// TIA Portal project "Bachelor_25.04.2025_1138" (V19)

(* hardware
DEVICE "S7-1500/ET200MP station_1"  S7-1500 station
   slot 0: "Rail_0"  Rack  6ES7 590-1***0-0AA0
   slot 0: "PM 70W 120/230VAC"  PM 70W 120/230VAC  6EP1332-4BA00
   slot 1: "PLC_1"  CPU 1511-1 PN  6ES7 511-1AK00-0AB0  V1.8
      slot 3: "CPU display_1"  6ES7591-1AA00-0AA0
      slot 32768: "PROFINET interface_1"  X1
         slot 32769: "Port_1"  X1 P1
         slot 32770: "Port_2"  X1 P2
   slot 2: "DI 16x24VDC HF_1"  DI 16x24VDC HF  6ES7 521-1BH00-0AB0  V1.0
   slot 3: "DQ 16x24VDC/0.5A ST_1"  DQ 16x24VDC/0.5A ST  6ES7 522-1BH00-0AB0  V2.0
   slot 4: "AI 8xU/I/RTD/TC ST_1"  AI 8xU/I/RTD/TC ST  6ES7 531-7KF00-0AB0  V1.0
   slot 5: "AQ 4xU/I ST_1"  AQ 4xU/I ST  6ES7 532-5HD00-0AB0  V1.0
   slot 6: "CM 1542-5_1"  CM 1542-5  6GK7 542-5DX00-0XE0  V2.0
*)

// ===== PLC "PLC_1"  CPU 1511-1 PN =====

VAR_GLOBAL   // PLC tag table "Default tag table"
   "F01" AT %I0.0 : Bool;
   "F02" AT %I0.1 : Bool;
   "F11" AT %I0.2 : Bool;
   "F12" AT %I0.3 : Bool;
   "S0" AT %I0.4 : Bool;
   "PU01_AUT" AT %I0.5 : Bool;
   "PU01_MAN" AT %I0.6 : Bool;
   "PU02_AUT" AT %I1.2 : Bool;
   "PU01_RUNNING" AT %I0.7 : Bool;
   "PU01_FAULT" AT %I1.0 : Bool;
   "PU01_SS" AT %I1.1 : Bool;
   "PU02_MAN" AT %I1.3 : Bool;
   "PU02_RUNNING" AT %I1.4 : Bool;
   "PU02_FAULT" AT %I1.5 : Bool;
   "PU02_SS" AT %I1.6 : Bool;
   "FV01_GB1" AT %I1.7 : Bool;
   "FV01_GB2" AT %I2.0 : Bool;
   "FV02_GB1" AT %I2.1 : Bool;
   "FV02_GB2" AT %I2.2 : Bool;
   "PU01_RUN" AT %Q0.0 : Bool;
   "PU02_RUN" AT %Q0.1 : Bool;
   "FV01_OPEN" AT %Q0.2 : Bool;
   "FV02_OPEN" AT %Q0.3 : Bool;
   "LT01_INT" AT %IW2 : Int;
   "FT01_INT" AT %IW10 : Int;
   "FT02_INT" AT %IW4 : Int;
   "PU01_INT" AT %QW2 : Int;
   "PU02_INT" AT %QW4 : Int;
   "M_F01" AT %M0.0 : Bool;
   "M_F02" AT %M0.1 : Bool;
   "M_F11" AT %M0.2 : Bool;
   "M_F12" AT %M0.3 : Bool;
   "M_S0" AT %M0.4 : Bool;
   "M_PU01_AUT" AT %M0.5 : Bool;
   "M_PU01_MAN" AT %M0.6 : Bool;
   "M_PU01_RUNNING" AT %M0.7 : Bool;
   "M_PU01_FAULT" AT %M2.0 : Bool;
   "M_PU01_SS" AT %M2.1 : Bool;
   "M_PU02_AUT" AT %M2.2 : Bool;
   "M_PU02_MAN" AT %M2.3 : Bool;
   "M_PU02_RUNNING" AT %M2.4 : Bool;
   "M_PU02_FAULT" AT %M2.5 : Bool;
   "M_PU02_SS" AT %M2.6 : Bool;
   "M_FV01_GB1" AT %M2.7 : Bool;
   "M_FV01_GB2" AT %M3.0 : Bool;
   "M_FV02_GB1" AT %M3.1 : Bool;
   "M_FV02_GB2" AT %M3.2 : Bool;
   "M_PU01_RUN" AT %M4.0 : Bool;
   "M_PU02_RUN" AT %M4.1 : Bool;
   "M_FV01" AT %M4.2 : Bool;
   "M_FV02" AT %M4.3 : Bool;
   "PU01_REAL" AT %MD100 : Real;
   "PU02_REAL" AT %MD104 : Real;
   "LT01_REAL" AT %MD108 : Real;
   "FT01_REAL" AT %MD1120 : Real;
   "FT02_REAL" AT %MD116 : Real;
   "RESET" AT %I2.3 : Bool;
   "Tag_1" AT %MW200 : Int;
   "Tag_21" AT %MW204 : Int;
   "Tag_22" AT %MW208 : Int;
   "Tag_23" AT %MW212 : Int;
   "Tag_24" AT %MW216 : Int;
   "BEST_HOURS" AT %MD50 : DInt;
   "OPTIMAL_HOUR" AT %M5.0 : Bool;
   "Tag_2" AT %MW300 : Word;
   "Tag_3" AT %MD320 : Real;
   "TRANSMIT" AT %I6.0 : "transmitter_dt";
   "CONTROLLER_STATE" AT %MW220 : Int;
   "M_PU01_AUT_SCADA" AT %M1000.0 : Bool;
   "M_PU01_MAN_SCADA" AT %M1.1 : Bool;
   "M_PU02_AUT_SCADA" AT %M1000.1 : Bool;
   "M_PU02_MAN_SCADA" AT %M3.4 : Bool;
   "ALWAYS HIGH" AT %M1.2 : Bool;
   "ALWAYS LOW" AT %M1.3 : Bool;
   "Clock_Byte" AT %MB6 : Byte;
   "Clock_10Hz" AT %M6.0 : Bool;
   "Clock_5Hz" AT %M6.1 : Bool;
   "Clock_2.5Hz" AT %M6.2 : Bool;
   "Clock_2Hz" AT %M6.3 : Bool;
   "Clock_1.25Hz" AT %M6.4 : Bool;
   "Clock_1Hz" AT %M6.5 : Bool;
   "Clock_0.625Hz" AT %M6.6 : Bool;
   "Clock_0.5Hz" AT %M6.7 : Bool;
   "BEST_HOURS_DAG2" AT %MD60 : DInt;
END_VAR

TYPE "transmitter_dt"
   STRUCT
      test_1 : Bool;
      test_2 : Bool;
      test_3 : Int;
   END_STRUCT;
END_TYPE

// folder: Data Blocks

DATA_BLOCK "FT02_DB"   // DB1
{ S7_Optimized_Access := 'FALSE' }
VERSION : 0.1
// stored: InstanceOfName Transmitter
"Transmitter"
BEGIN
   t_sp_hh_pct := 100.0;
   t_sp_h_pct := 100.0;
   t_sp_l_pct := 0.0;
   t_sp_ll_pct := 0.0;
   t_sp_scale_high_pct := 100.0;
END_DATA_BLOCK

DATA_BLOCK "Cascade Regulator_DB"   // DB2
{ S7_Optimized_Access := 'FALSE' }
VERSION : 0.1
// stored: InstanceOfName Cascade Regulator
"Cascade Regulator"
BEGIN
END_DATA_BLOCK

DATA_BLOCK "PU02_DB"   // DB3
{ S7_Optimized_Access := 'FALSE' }
VERSION : 0.1
// stored: InstanceOfName Pump
"Pump"
BEGIN
END_DATA_BLOCK

DATA_BLOCK "LT01_DB"   // DB5
{ S7_Optimized_Access := 'FALSE' }
VERSION : 0.1
// stored: InstanceOfName Transmitter
"Transmitter"
BEGIN
   t_hys := 1;
   t_sp_hh_pct := 95.0;
   t_sp_h_pct := 90.0;
   t_sp_l_pct := 30.0;
   t_sp_ll_pct := 25.0;
   t_sp_scale_high_pct := 100.0;
   t_sp_scale_high_sca := 4.0;
   t_sp_hh_sca := 3.8;
   t_sp_h_sca := 3.6;
   t_sp_l_sca := 0.9;
   t_sp_ll_sca := 0.6;
END_DATA_BLOCK

DATA_BLOCK "FT01_DB"   // DB6
{ S7_Optimized_Access := 'FALSE' }
VERSION : 0.1
// stored: InstanceOfName Transmitter
"Transmitter"
BEGIN
   t_sp_hh_pct := 100.0;
   t_sp_h_pct := 100.0;
   t_sp_l_pct := 0.0;
   t_sp_ll_pct := 0.0;
   t_sp_scale_high_pct := 100.0;
   t_sp_scale_high_sca := 50.0;
   t_sp_hh_sca := 50.0;
   t_sp_h_sca := 50.0;
END_DATA_BLOCK

DATA_BLOCK "Control_block_DB"   // DB7
{ S7_Optimized_Access := 'FALSE' }
VERSION : 0.1
// stored: InstanceOfName Control block
"Control block"
BEGIN
END_DATA_BLOCK

DATA_BLOCK "PU01_DB"   // DB14
{ S7_Optimized_Access := 'FALSE' }
VERSION : 0.1
// stored: InstanceOfName Pump
"Pump"
BEGIN
END_DATA_BLOCK

DATA_BLOCK "Check optimal hour 48h_DB"   // DB29
{ S7_Optimized_Access := 'TRUE' }
VERSION : 0.1
// stored: InstanceOfName Check optimal hour 48h
"Check optimal hour 48h"
BEGIN
END_DATA_BLOCK

// folder: System blocks/Program resources

DATA_BLOCK "IEC_Timer_0_DB"   // DB4
{ S7_Optimized_Access := 'TRUE' }
AUTHOR : Simatic
FAMILY : IEC
NAME : IEC_TMR
VERSION : 1.0
// stored: InstanceOfName IEC_TIMER
"IEC_TIMER"
BEGIN
END_DATA_BLOCK

DATA_BLOCK "t_alarm_hys"   // DB8
{ S7_Optimized_Access := 'TRUE' }
AUTHOR : Simatic
FAMILY : IEC
NAME : IEC_TMR
VERSION : 1.0
// stored: InstanceOfName IEC_TIMER
"IEC_TIMER"
BEGIN
END_DATA_BLOCK

DATA_BLOCK "IEC_Timer_0_DB_2"   // DB11
{ S7_Optimized_Access := 'TRUE' }
AUTHOR : Simatic
FAMILY : IEC
NAME : IEC_TMR
VERSION : 1.0
// stored: InstanceOfName IEC_TIMER
"IEC_TIMER"
BEGIN
END_DATA_BLOCK

DATA_BLOCK "t_alarm_hh"   // DB12
{ S7_Optimized_Access := 'TRUE' }
AUTHOR : Simatic
FAMILY : IEC
NAME : IEC_TMR
VERSION : 1.0
// stored: InstanceOfName IEC_TIMER
"IEC_TIMER"
BEGIN
END_DATA_BLOCK

DATA_BLOCK "t_alarm_h"   // DB13
{ S7_Optimized_Access := 'TRUE' }
AUTHOR : Simatic
FAMILY : IEC
NAME : IEC_TMR
VERSION : 1.0
// stored: InstanceOfName IEC_TIMER
"IEC_TIMER"
BEGIN
END_DATA_BLOCK

DATA_BLOCK "t_alarm_l"   // DB15
{ S7_Optimized_Access := 'TRUE' }
AUTHOR : Simatic
FAMILY : IEC
NAME : IEC_TMR
VERSION : 1.0
// stored: InstanceOfName IEC_TIMER
"IEC_TIMER"
BEGIN
END_DATA_BLOCK

DATA_BLOCK "t_alarm_ll"   // DB16
{ S7_Optimized_Access := 'TRUE' }
AUTHOR : Simatic
FAMILY : IEC
NAME : IEC_TMR
VERSION : 1.0
// stored: InstanceOfName IEC_TIMER
"IEC_TIMER"
BEGIN
END_DATA_BLOCK

DATA_BLOCK "t_alarm_range"   // DB17
{ S7_Optimized_Access := 'TRUE' }
AUTHOR : Simatic
FAMILY : IEC
NAME : IEC_TMR
VERSION : 1.0
// stored: InstanceOfName IEC_TIMER
"IEC_TIMER"
BEGIN
END_DATA_BLOCK

DATA_BLOCK "p_alarm_fv"   // DB18
{ S7_Optimized_Access := 'TRUE' }
AUTHOR : Simatic
FAMILY : IEC
NAME : IEC_TMR
VERSION : 1.0
// stored: InstanceOfName IEC_TIMER
"IEC_TIMER"
BEGIN
END_DATA_BLOCK

DATA_BLOCK "p_alarm_vfd"   // DB19
{ S7_Optimized_Access := 'TRUE' }
AUTHOR : Simatic
FAMILY : IEC
NAME : IEC_TMR
VERSION : 1.0
// stored: InstanceOfName IEC_TIMER
"IEC_TIMER"
BEGIN
END_DATA_BLOCK

DATA_BLOCK "p_alarm_tmp"   // DB20
{ S7_Optimized_Access := 'TRUE' }
AUTHOR : Simatic
FAMILY : IEC
NAME : IEC_TMR
VERSION : 1.0
// stored: InstanceOfName IEC_TIMER
"IEC_TIMER"
BEGIN
END_DATA_BLOCK

DATA_BLOCK "p_alarm_moi"   // DB21
{ S7_Optimized_Access := 'TRUE' }
AUTHOR : Simatic
FAMILY : IEC
NAME : IEC_TMR
VERSION : 1.0
// stored: InstanceOfName IEC_TIMER
"IEC_TIMER"
BEGIN
END_DATA_BLOCK

DATA_BLOCK "p_alarm"   // DB22
{ S7_Optimized_Access := 'TRUE' }
AUTHOR : Simatic
FAMILY : IEC
NAME : IEC_TMR
VERSION : 1.0
// stored: InstanceOfName IEC_TIMER
"IEC_TIMER"
BEGIN
END_DATA_BLOCK

DATA_BLOCK "Input Error"   // DB23
{ S7_Optimized_Access := 'TRUE' }
AUTHOR : Simatic
FAMILY : IEC
NAME : IEC_TMR
VERSION : 1.0
// stored: InstanceOfName IEC_TIMER
"IEC_TIMER"
BEGIN
END_DATA_BLOCK

DATA_BLOCK "Tuning Error"   // DB24
{ S7_Optimized_Access := 'TRUE' }
AUTHOR : Simatic
FAMILY : IEC
NAME : IEC_TMR
VERSION : 1.0
// stored: InstanceOfName IEC_TIMER
"IEC_TIMER"
BEGIN
END_DATA_BLOCK

DATA_BLOCK "Setpoint Error"   // DB25
{ S7_Optimized_Access := 'TRUE' }
AUTHOR : Simatic
FAMILY : IEC
NAME : IEC_TMR
VERSION : 1.0
// stored: InstanceOfName IEC_TIMER
"IEC_TIMER"
BEGIN
END_DATA_BLOCK

DATA_BLOCK "ManualValue Error"   // DB26
{ S7_Optimized_Access := 'TRUE' }
AUTHOR : Simatic
FAMILY : IEC
NAME : IEC_TMR
VERSION : 1.0
// stored: InstanceOfName IEC_TIMER
"IEC_TIMER"
BEGIN
END_DATA_BLOCK

DATA_BLOCK "General Error"   // DB27
{ S7_Optimized_Access := 'TRUE' }
AUTHOR : Simatic
FAMILY : IEC
NAME : IEC_TMR
VERSION : 1.0
// stored: InstanceOfName IEC_TIMER
"IEC_TIMER"
BEGIN
END_DATA_BLOCK

DATA_BLOCK "Regulator Error"   // DB28
{ S7_Optimized_Access := 'TRUE' }
AUTHOR : Simatic
FAMILY : IEC
NAME : IEC_TMR
VERSION : 1.0
// stored: InstanceOfName IEC_TIMER
"IEC_TIMER"
BEGIN
END_DATA_BLOCK

DATA_BLOCK "CV_unmod"   // DB30
{ S7_Optimized_Access := 'TRUE' }
AUTHOR : Simatic
FAMILY : IEC
NAME : IEC_TMR
VERSION : 1.0
// stored: InstanceOfName IEC_TIMER
"IEC_TIMER"
BEGIN
END_DATA_BLOCK

DATA_BLOCK "Timer"   // DB31
{ S7_Optimized_Access := 'TRUE' }
AUTHOR : Simatic
FAMILY : IEC
NAME : IEC_TMR
VERSION : 1.0
// stored: InstanceOfName IEC_TIMER
"IEC_TIMER"
BEGIN
END_DATA_BLOCK

DATA_BLOCK "p_alarm_flow"   // DB32
{ S7_Optimized_Access := 'TRUE' }
AUTHOR : Simatic
FAMILY : IEC
NAME : IEC_TMR
VERSION : 1.0
// stored: InstanceOfName IEC_TIMER
"IEC_TIMER"
BEGIN
END_DATA_BLOCK

// folder: (top level)

FUNCTION_BLOCK "Control block"   // FB1, LAD
{ S7_Optimized_Access := 'FALSE' }
VERSION : 0.1
   VAR_INPUT
      pu01_aut : Bool;
      pu01_aut_scada : Bool := true;
      pu01_man : Bool;
      pu01_man_scada : Bool;
      pu01_mv : Real;
      pu01_fault : Bool;
      pu02_aut : Bool;
      pu02_aut_scada : Bool := true;
      pu02_man : Bool;
      pu02_man_scada : Bool;
      pu02_mv : Real;
      pu02_fault : Bool;
      setpoint_high : Real;
      setpoint_low : Real;
      controller_cv : Real;
      pump_time : Time := T#30s;
   END_VAR
   VAR_OUTPUT
      controller_state : Int;
      controller_mv : Real;
   END_VAR
   VAR_IN_OUT
      pu01_run : Bool;
      pu01_running : Bool;
      pu02_run : Bool;
      pu02_running : Bool;
   END_VAR
   VAR
      "pu01 is in aut" : Bool;
      "pu01 is in man" : Bool;
      "pu02 is in aut" : Bool;
      "pu02 is in man" : Bool;
      yup : Int;
      yupper : Bool;
      n_trig_0 : Bool;
      n_trig_1 : Bool;
      n_trig_2 : Bool;
      n_trig_3 : Bool;
      pu01_timer : Time := T#30s;
      pu02_timer : Time := T#40s;
   END_VAR
   VAR_TEMP   // added for the SCL form of the ladder/FBD networks
      _w1 : Bool;
      _w2 : Bool;
   END_VAR
BEGIN

REGION Network 1: PU01 Automatic
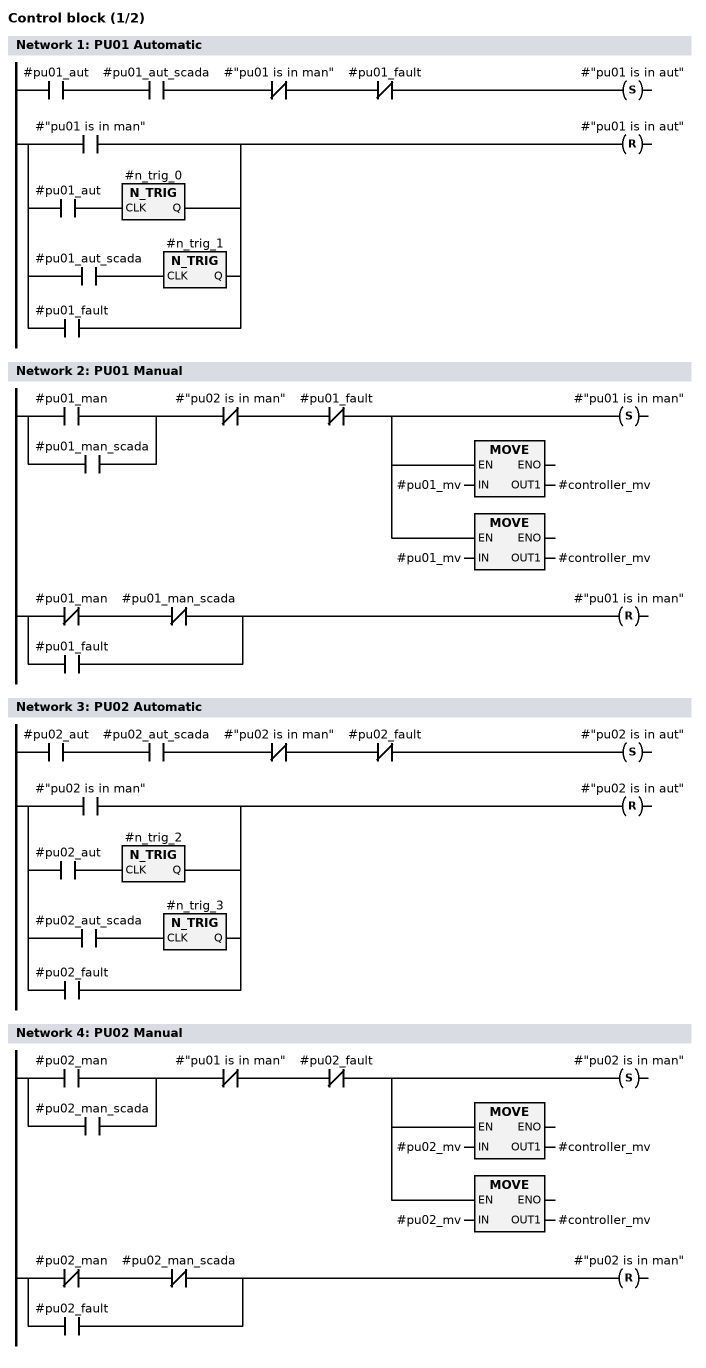
   RUNG wire#powerrail
      Contact( #pu01_aut )
      Contact( #pu01_aut_scada )
      I_Contact( #"pu01 is in man" )
      I_Contact( #pu01_fault )
      S_Coil( #"pu01 is in aut" )
   END_RUNG
   RUNG wire#powerrail
      Contact( #"pu01 is in man" )
      wire#w1
      R_Coil( #"pu01 is in aut" )
   END_RUNG
   RUNG wire#powerrail
      Contact( #pu01_aut )
      N_Trig( #n_trig_0 )
   END_RUNG wire#w1
   RUNG wire#powerrail
      Contact( #pu01_aut_scada )
      N_Trig( #n_trig_1 )
   END_RUNG wire#w1
   RUNG wire#powerrail
      Contact( #pu01_fault )
   END_RUNG wire#w1
   // the same network as SCL:
   IF #pu01_aut AND #pu01_aut_scada AND NOT #"pu01 is in man" AND NOT #pu01_fault THEN
       #"pu01 is in aut" := TRUE;
   END_IF;
   #_w1 := NOT #pu01_aut AND #n_trig_0;   // falling edge
   #n_trig_0 := #pu01_aut;
   #_w2 := NOT #pu01_aut_scada AND #n_trig_1;   // falling edge
   #n_trig_1 := #pu01_aut_scada;
   IF #"pu01 is in man" OR #_w1 OR #_w2 OR #pu01_fault THEN #"pu01 is in aut" := FALSE; END_IF;
END_REGION

REGION Network 2: PU01 Manual
   RUNG wire#powerrail
      Contact( #pu01_man )
      wire#w1
      I_Contact( #"pu02 is in man" )
      I_Contact( #pu01_fault )
      wire#w2
      S_Coil( #"pu01 is in man" )
   END_RUNG
   RUNG wire#powerrail
      Contact( #pu01_man_scada )
   END_RUNG wire#w1
   RUNG wire#w2
      Move(in := #pu01_mv, out1 => #controller_mv)
   END_RUNG
   RUNG wire#w2
      Move(in := #pu01_mv, out1 => #controller_mv)
   END_RUNG
   RUNG wire#powerrail
      I_Contact( #pu01_man )
      I_Contact( #pu01_man_scada )
      wire#w3
      R_Coil( #"pu01 is in man" )
   END_RUNG
   RUNG wire#powerrail
      Contact( #pu01_fault )
   END_RUNG wire#w3
   // the same network as SCL:
   IF (#pu01_man OR #pu01_man_scada) AND NOT #"pu02 is in man" AND NOT #pu01_fault THEN
       #"pu01 is in man" := TRUE;
       #controller_mv := #pu01_mv;
       #controller_mv := #pu01_mv;
   END_IF;
   IF (NOT #pu01_man AND NOT #pu01_man_scada) OR #pu01_fault THEN #"pu01 is in man" := FALSE; END_IF;
END_REGION

REGION Network 3: PU02 Automatic
   RUNG wire#powerrail
      Contact( #pu02_aut )
      Contact( #pu02_aut_scada )
      I_Contact( #"pu02 is in man" )
      I_Contact( #pu02_fault )
      S_Coil( #"pu02 is in aut" )
   END_RUNG
   RUNG wire#powerrail
      Contact( #"pu02 is in man" )
      wire#w1
      R_Coil( #"pu02 is in aut" )
   END_RUNG
   RUNG wire#powerrail
      Contact( #pu02_aut )
      N_Trig( #n_trig_2 )
   END_RUNG wire#w1
   RUNG wire#powerrail
      Contact( #pu02_aut_scada )
      N_Trig( #n_trig_3 )
   END_RUNG wire#w1
   RUNG wire#powerrail
      Contact( #pu02_fault )
   END_RUNG wire#w1
   // the same network as SCL:
   IF #pu02_aut AND #pu02_aut_scada AND NOT #"pu02 is in man" AND NOT #pu02_fault THEN
       #"pu02 is in aut" := TRUE;
   END_IF;
   #_w1 := NOT #pu02_aut AND #n_trig_2;   // falling edge
   #n_trig_2 := #pu02_aut;
   #_w2 := NOT #pu02_aut_scada AND #n_trig_3;   // falling edge
   #n_trig_3 := #pu02_aut_scada;
   IF #"pu02 is in man" OR #_w1 OR #_w2 OR #pu02_fault THEN #"pu02 is in aut" := FALSE; END_IF;
END_REGION

REGION Network 4: PU02 Manual
   RUNG wire#powerrail
      Contact( #pu02_man )
      wire#w1
      I_Contact( #"pu01 is in man" )
      I_Contact( #pu02_fault )
      wire#w2
      S_Coil( #"pu02 is in man" )
   END_RUNG
   RUNG wire#powerrail
      Contact( #pu02_man_scada )
   END_RUNG wire#w1
   RUNG wire#w2
      Move(in := #pu02_mv, out1 => #controller_mv)
   END_RUNG
   RUNG wire#w2
      Move(in := #pu02_mv, out1 => #controller_mv)
   END_RUNG
   RUNG wire#powerrail
      I_Contact( #pu02_man )
      I_Contact( #pu02_man_scada )
      wire#w3
      R_Coil( #"pu02 is in man" )
   END_RUNG
   RUNG wire#powerrail
      Contact( #pu02_fault )
   END_RUNG wire#w3
   // the same network as SCL:
   IF (#pu02_man OR #pu02_man_scada) AND NOT #"pu01 is in man" AND NOT #pu02_fault THEN
       #"pu02 is in man" := TRUE;
       #controller_mv := #pu02_mv;
       #controller_mv := #pu02_mv;
   END_IF;
   IF (NOT #pu02_man AND NOT #pu02_man_scada) OR #pu02_fault THEN #"pu02 is in man" := FALSE; END_IF;
END_REGION

REGION Network 5: Controller Auto
   // Sets the Controller in auto if it can.
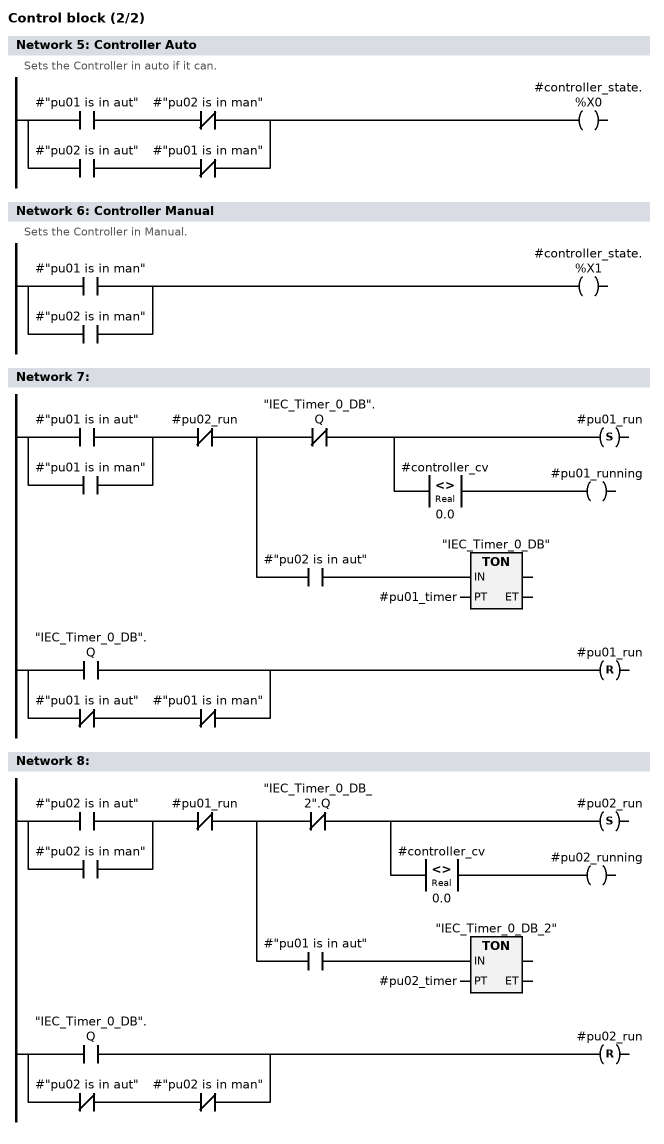
   RUNG wire#powerrail
      Contact( #"pu01 is in aut" )
      I_Contact( #"pu02 is in man" )
      wire#w1
      Coil( #controller_state.%X0 )
   END_RUNG
   RUNG wire#powerrail
      Contact( #"pu02 is in aut" )
      I_Contact( #"pu01 is in man" )
   END_RUNG wire#w1
   // the same network as SCL:
   #controller_state.%X0 := (#"pu01 is in aut" AND NOT #"pu02 is in man") OR (#"pu02 is in aut" AND NOT #"pu01 is in man");
END_REGION

REGION Network 6: Controller Manual
   // Sets the Controller in Manual.
   RUNG wire#powerrail
      Contact( #"pu01 is in man" )
      wire#w1
      Coil( #controller_state.%X1 )
   END_RUNG
   RUNG wire#powerrail
      Contact( #"pu02 is in man" )
   END_RUNG wire#w1
   // the same network as SCL:
   #controller_state.%X1 := #"pu01 is in man" OR #"pu02 is in man";
END_REGION

REGION Network 7
   #_w1 := (#"pu01 is in aut" OR #"pu01 is in man") AND NOT #pu02_run;
   #_w2 := #_w1 AND NOT "IEC_Timer_0_DB".Q;
   IF #_w2 THEN #pu01_run := TRUE; END_IF;
   #pu01_running := #_w2 AND (#controller_cv <> 0.0);
   "IEC_Timer_0_DB".TON(IN := #_w1 AND #"pu02 is in aut", PT := #pu01_timer);
   IF "IEC_Timer_0_DB".Q OR (NOT #"pu01 is in aut" AND NOT #"pu01 is in man") THEN
       #pu01_run := FALSE;
   END_IF;
END_REGION

REGION Network 8
   #_w1 := (#"pu02 is in aut" OR #"pu02 is in man") AND NOT #pu01_run;
   #_w2 := #_w1 AND NOT "IEC_Timer_0_DB_2".Q;
   IF #_w2 THEN #pu02_run := TRUE; END_IF;
   #pu02_running := #_w2 AND (#controller_cv <> 0.0);
   "IEC_Timer_0_DB_2".TON(IN := #_w1 AND #"pu01 is in aut", PT := #pu02_timer);
   IF "IEC_Timer_0_DB".Q OR (NOT #"pu02 is in aut" AND NOT #"pu02 is in man") THEN
       #pu02_run := FALSE;
   END_IF;
END_REGION
END_FUNCTION_BLOCK

FUNCTION "Convert Analog Values" : Void   // FC1, LAD
{ S7_Optimized_Access := 'TRUE' }
VERSION : 0.1
   VAR_INPUT
      lt01_int : Int;
      ft01_int : Int;
      ft02_int : Int;
      pu01_real : Real;
      pu02_real : Real;
   END_VAR
   VAR_OUTPUT
      lt01_real : Real;
      ft01_real : Real;
      ft02_real : Real;
      pu01_int : Int;
      pu02_int : Int;
   END_VAR
   VAR_TEMP
      lt01_temp : Real;
      ft01_temp : Real;
      ft02_temp : Real;
      pu01_temp : Real;
      pu02_temp : Real;
   END_VAR
BEGIN

REGION Network 1: Level Transmitter 01
   // Level Transmitter in the pool
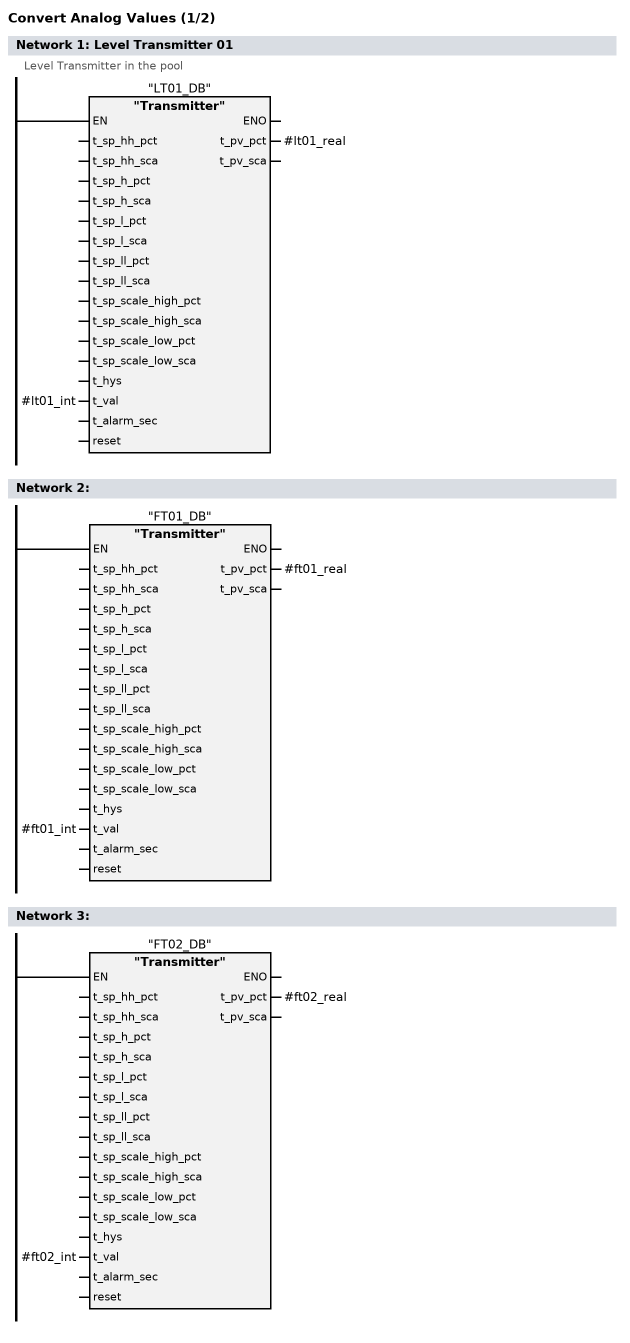
   RUNG wire#powerrail
      "LT01_DB"(t_sp_hh_pct :=, t_sp_hh_sca :=, t_sp_h_pct :=, t_sp_h_sca :=, t_sp_l_pct :=, t_sp_l_sca :=, t_sp_ll_pct :=, t_sp_ll_sca :=, t_sp_scale_high_pct :=, t_sp_scale_high_sca :=, t_sp_scale_low_pct :=, t_sp_scale_low_sca :=, t_hys :=, t_val := #lt01_int, t_alarm_sec :=, reset :=, t_pv_pct => #lt01_real, t_pv_sca =>)
   END_RUNG
   // the same network as SCL:
   "LT01_DB"(t_val := #lt01_int, t_pv_pct => #lt01_real);   // "Transmitter"
END_REGION

REGION Network 2
   RUNG wire#powerrail
      "FT01_DB"(t_sp_hh_pct :=, t_sp_hh_sca :=, t_sp_h_pct :=, t_sp_h_sca :=, t_sp_l_pct :=, t_sp_l_sca :=, t_sp_ll_pct :=, t_sp_ll_sca :=, t_sp_scale_high_pct :=, t_sp_scale_high_sca :=, t_sp_scale_low_pct :=, t_sp_scale_low_sca :=, t_hys :=, t_val := #ft01_int, t_alarm_sec :=, reset :=, t_pv_pct => #ft01_real, t_pv_sca =>)
   END_RUNG
   // the same network as SCL:
   "FT01_DB"(t_val := #ft01_int, t_pv_pct => #ft01_real);   // "Transmitter"
END_REGION

REGION Network 3
   RUNG wire#powerrail
      "FT02_DB"(t_sp_hh_pct :=, t_sp_hh_sca :=, t_sp_h_pct :=, t_sp_h_sca :=, t_sp_l_pct :=, t_sp_l_sca :=, t_sp_ll_pct :=, t_sp_ll_sca :=, t_sp_scale_high_pct :=, t_sp_scale_high_sca :=, t_sp_scale_low_pct :=, t_sp_scale_low_sca :=, t_hys :=, t_val := #ft02_int, t_alarm_sec :=, reset :=, t_pv_pct => #ft02_real, t_pv_sca =>)
   END_RUNG
   // the same network as SCL:
   "FT02_DB"(t_val := #ft02_int, t_pv_pct => #ft02_real);   // "Transmitter"
END_REGION

REGION Network 4: Signal til frekvensomformeren som tilhører PU01
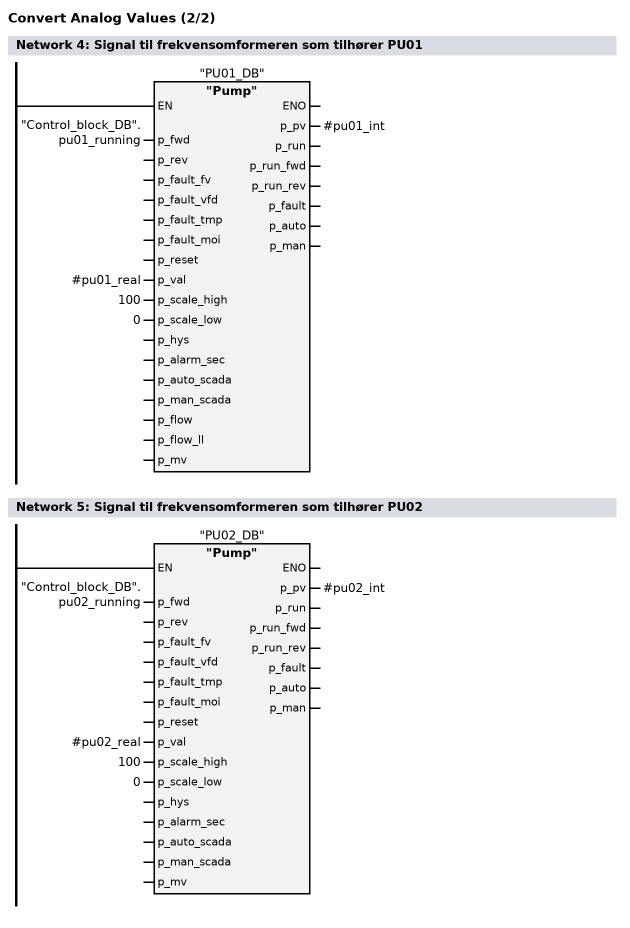
   RUNG wire#powerrail
      "PU01_DB"(p_fwd := "Control_block_DB".pu01_running, p_rev :=, p_fault_fv :=, p_fault_vfd :=, p_fault_tmp :=, p_fault_moi :=, p_reset :=, p_val := #pu01_real, p_scale_high := 100, p_scale_low := 0, p_hys :=, p_alarm_sec :=, p_auto_scada :=, p_man_scada :=, p_flow :=, p_flow_ll :=, p_mv :=, p_pv => #pu01_int, p_run =>, p_run_fwd =>, p_run_rev =>, p_fault =>, p_auto =>, p_man =>)
   END_RUNG
   // the same network as SCL:
   "PU01_DB"(p_fwd := "Control_block_DB".pu01_running,   // "Pump"
             p_val := #pu01_real,
             p_scale_high := 100,
             p_scale_low := 0,
             p_pv => #pu01_int);
END_REGION

REGION Network 5: Signal til frekvensomformeren som tilhører PU02
   RUNG wire#powerrail
      "PU02_DB"(p_fwd := "Control_block_DB".pu02_running, p_rev :=, p_fault_fv :=, p_fault_vfd :=, p_fault_tmp :=, p_fault_moi :=, p_reset :=, p_val := #pu02_real, p_scale_high := 100, p_scale_low := 0, p_hys :=, p_alarm_sec :=, p_auto_scada :=, p_man_scada :=, p_mv :=, p_pv => #pu02_int, p_run =>, p_run_fwd =>, p_run_rev =>, p_fault =>, p_auto =>, p_man =>)
   END_RUNG
   // the same network as SCL:
   "PU02_DB"(p_fwd := "Control_block_DB".pu02_running,   // "Pump"
             p_val := #pu02_real,
             p_scale_high := 100,
             p_scale_low := 0,
             p_pv => #pu02_int);
END_REGION
END_FUNCTION

FUNCTION "Input Mapping" : Void   // FC3, LAD
TITLE = Convert I/O to M
{ S7_Optimized_Access := 'TRUE' }
VERSION : 0.1
BEGIN

REGION Network 1: Digital Inputs
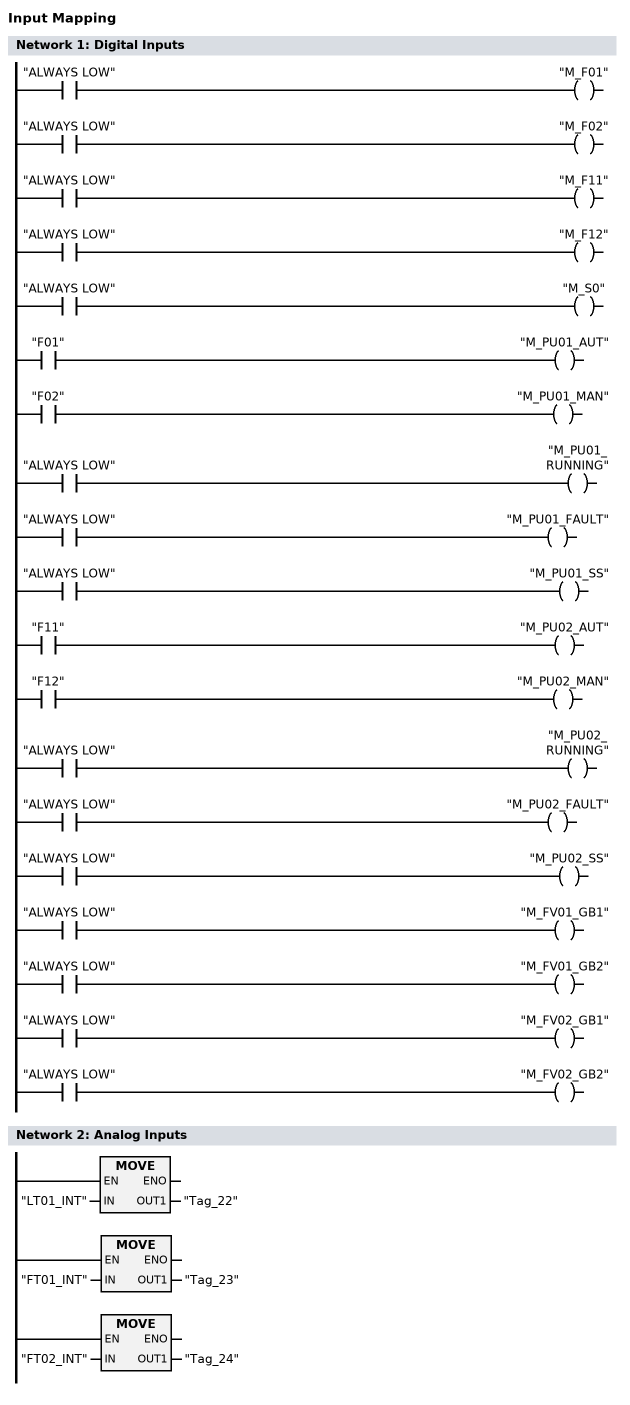
   RUNG wire#powerrail
      Contact( "ALWAYS LOW" )
      Coil( "M_F01" )
   END_RUNG
   RUNG wire#powerrail
      Contact( "ALWAYS LOW" )
      Coil( "M_F02" )
   END_RUNG
   RUNG wire#powerrail
      Contact( "ALWAYS LOW" )
      Coil( "M_F11" )
   END_RUNG
   RUNG wire#powerrail
      Contact( "ALWAYS LOW" )
      Coil( "M_F12" )
   END_RUNG
   RUNG wire#powerrail
      Contact( "ALWAYS LOW" )
      Coil( "M_S0" )
   END_RUNG
   RUNG wire#powerrail
      Contact( "F01" )
      Coil( "M_PU01_AUT" )
   END_RUNG
   RUNG wire#powerrail
      Contact( "F02" )
      Coil( "M_PU01_MAN" )
   END_RUNG
   RUNG wire#powerrail
      Contact( "ALWAYS LOW" )
      Coil( "M_PU01_RUNNING" )
   END_RUNG
   RUNG wire#powerrail
      Contact( "ALWAYS LOW" )
      Coil( "M_PU01_FAULT" )
   END_RUNG
   RUNG wire#powerrail
      Contact( "ALWAYS LOW" )
      Coil( "M_PU01_SS" )
   END_RUNG
   RUNG wire#powerrail
      Contact( "F11" )
      Coil( "M_PU02_AUT" )
   END_RUNG
   RUNG wire#powerrail
      Contact( "F12" )
      Coil( "M_PU02_MAN" )
   END_RUNG
   RUNG wire#powerrail
      Contact( "ALWAYS LOW" )
      Coil( "M_PU02_RUNNING" )
   END_RUNG
   RUNG wire#powerrail
      Contact( "ALWAYS LOW" )
      Coil( "M_PU02_FAULT" )
   END_RUNG
   RUNG wire#powerrail
      Contact( "ALWAYS LOW" )
      Coil( "M_PU02_SS" )
   END_RUNG
   RUNG wire#powerrail
      Contact( "ALWAYS LOW" )
      Coil( "M_FV01_GB1" )
   END_RUNG
   RUNG wire#powerrail
      Contact( "ALWAYS LOW" )
      Coil( "M_FV01_GB2" )
   END_RUNG
   RUNG wire#powerrail
      Contact( "ALWAYS LOW" )
      Coil( "M_FV02_GB1" )
   END_RUNG
   RUNG wire#powerrail
      Contact( "ALWAYS LOW" )
      Coil( "M_FV02_GB2" )
   END_RUNG
   // the same network as SCL:
   "M_F01" := "ALWAYS LOW";
   "M_F02" := "ALWAYS LOW";
   "M_F11" := "ALWAYS LOW";
   "M_F12" := "ALWAYS LOW";
   "M_S0" := "ALWAYS LOW";
   "M_PU01_AUT" := "F01";
   "M_PU01_MAN" := "F02";
   "M_PU01_RUNNING" := "ALWAYS LOW";
   "M_PU01_FAULT" := "ALWAYS LOW";
   "M_PU01_SS" := "ALWAYS LOW";
   "M_PU02_AUT" := "F11";
   "M_PU02_MAN" := "F12";
   "M_PU02_RUNNING" := "ALWAYS LOW";
   "M_PU02_FAULT" := "ALWAYS LOW";
   "M_PU02_SS" := "ALWAYS LOW";
   "M_FV01_GB1" := "ALWAYS LOW";
   "M_FV01_GB2" := "ALWAYS LOW";
   "M_FV02_GB1" := "ALWAYS LOW";
   "M_FV02_GB2" := "ALWAYS LOW";
END_REGION

REGION Network 2: Analog Inputs
   RUNG wire#powerrail
      Move(in := "LT01_INT", out1 => "Tag_22")
   END_RUNG
   RUNG wire#powerrail
      Move(in := "FT01_INT", out1 => "Tag_23")
   END_RUNG
   RUNG wire#powerrail
      Move(in := "FT02_INT", out1 => "Tag_24")
   END_RUNG
   // the same network as SCL:
   "Tag_22" := "LT01_INT";
   "Tag_23" := "FT01_INT";
   "Tag_24" := "FT02_INT";
END_REGION
END_FUNCTION

FUNCTION "Output Mapping" : Void   // FC4, LAD
{ S7_Optimized_Access := 'TRUE' }
VERSION : 0.1
BEGIN

REGION Network 1: Digital Outputs
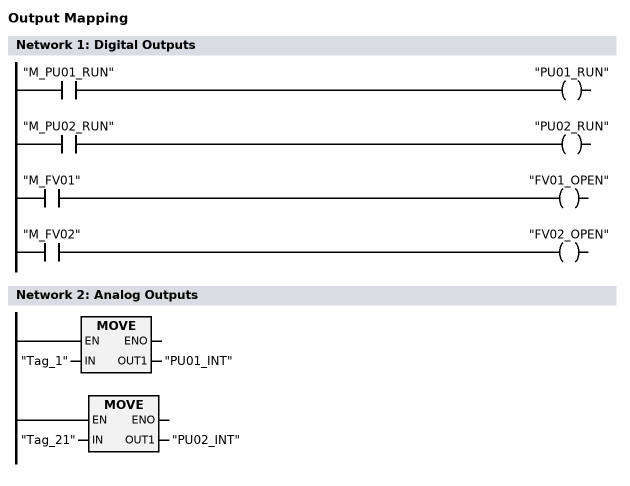
   RUNG wire#powerrail
      Contact( "M_PU01_RUN" )
      Coil( "PU01_RUN" )
   END_RUNG
   RUNG wire#powerrail
      Contact( "M_PU02_RUN" )
      Coil( "PU02_RUN" )
   END_RUNG
   RUNG wire#powerrail
      Contact( "M_FV01" )
      Coil( "FV01_OPEN" )
   END_RUNG
   RUNG wire#powerrail
      Contact( "M_FV02" )
      Coil( "FV02_OPEN" )
   END_RUNG
   // the same network as SCL:
   "PU01_RUN" := "M_PU01_RUN";
   "PU02_RUN" := "M_PU02_RUN";
   "FV01_OPEN" := "M_FV01";
   "FV02_OPEN" := "M_FV02";
END_REGION

REGION Network 2: Analog Outputs
   RUNG wire#powerrail
      Move(in := "Tag_1", out1 => "PU01_INT")
   END_RUNG
   RUNG wire#powerrail
      Move(in := "Tag_21", out1 => "PU02_INT")
   END_RUNG
   // the same network as SCL:
   "PU01_INT" := "Tag_1";
   "PU02_INT" := "Tag_21";
END_REGION
END_FUNCTION

ORGANIZATION_BLOCK "Main"   // OB1, LAD, ProgramCycle
TITLE = "Main Program Sweep (Cycle)"
{ S7_Optimized_Access := 'TRUE' }
VERSION : 0.1
   VAR_INPUT
      Initial_Call : Bool;   // Initial call of this OB
      Remanence : Bool;   // =True, if remanent data are available
   END_VAR
BEGIN

REGION Network 1
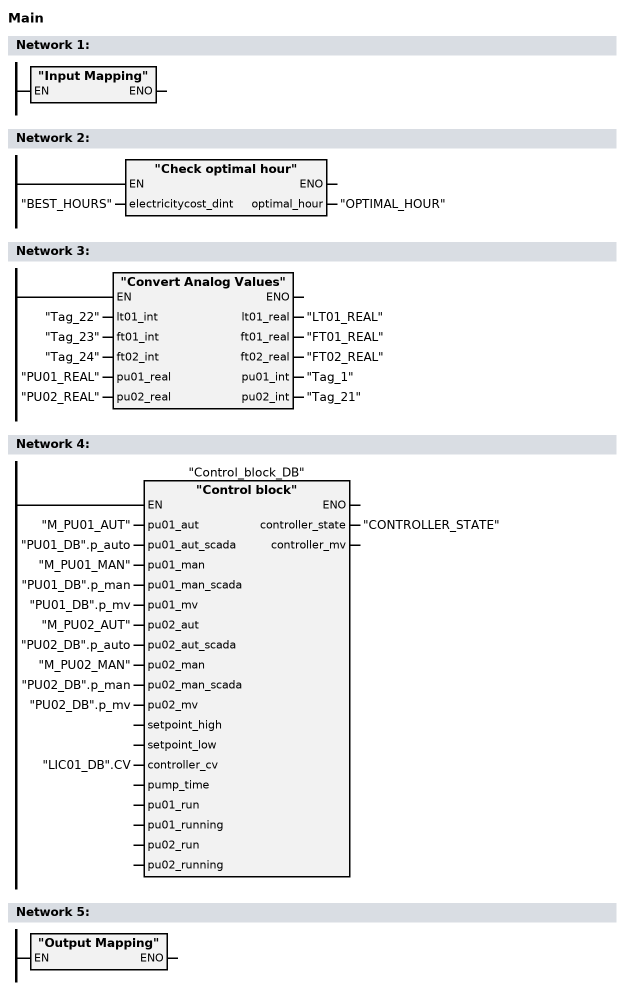
   RUNG wire#powerrail
      "Input Mapping"()
   END_RUNG
   // the same network as SCL:
   "Input Mapping"();
END_REGION

REGION Network 2
   RUNG wire#powerrail
      "Check optimal hour"(electricitycost_dint := "BEST_HOURS", optimal_hour => "OPTIMAL_HOUR")
   END_RUNG
   // the same network as SCL:
   "Check optimal hour"(electricitycost_dint := "BEST_HOURS", optimal_hour => "OPTIMAL_HOUR");
END_REGION

REGION Network 3
   RUNG wire#powerrail
      "Convert Analog Values"(lt01_int := "Tag_22", ft01_int := "Tag_23", ft02_int := "Tag_24", pu01_real := "PU01_REAL", pu02_real := "PU02_REAL", lt01_real => "LT01_REAL", ft01_real => "FT01_REAL", ft02_real => "FT02_REAL", pu01_int => "Tag_1", pu02_int => "Tag_21")
   END_RUNG
   // the same network as SCL:
   "Convert Analog Values"(lt01_int := "Tag_22",
                           ft01_int := "Tag_23",
                           ft02_int := "Tag_24",
                           pu01_real := "PU01_REAL",
                           pu02_real := "PU02_REAL",
                           lt01_real => "LT01_REAL",
                           ft01_real => "FT01_REAL",
                           ft02_real => "FT02_REAL",
                           pu01_int => "Tag_1",
                           pu02_int => "Tag_21");
END_REGION

REGION Network 4
   RUNG wire#powerrail
      "Control_block_DB"(pu01_aut := "M_PU01_AUT", pu01_aut_scada := "PU01_DB".p_auto, pu01_man := "M_PU01_MAN", pu01_man_scada := "PU01_DB".p_man, pu01_mv := "PU01_DB".p_mv, pu02_aut := "M_PU02_AUT", pu02_aut_scada := "PU02_DB".p_auto, pu02_man := "M_PU02_MAN", pu02_man_scada := "PU02_DB".p_man, pu02_mv := "PU02_DB".p_mv, setpoint_high :=, setpoint_low :=, controller_cv := "LIC01_DB".CV, pump_time :=, pu01_run :=, pu01_running :=, pu02_run :=, pu02_running :=, controller_state => "CONTROLLER_STATE", controller_mv =>)
   END_RUNG
   // the same network as SCL:
   "Control_block_DB"(pu01_aut := "M_PU01_AUT",   // "Control block"
                      pu01_aut_scada := "PU01_DB".p_auto,
                      pu01_man := "M_PU01_MAN",
                      pu01_man_scada := "PU01_DB".p_man,
                      pu01_mv := "PU01_DB".p_mv,
                      pu02_aut := "M_PU02_AUT",
                      pu02_aut_scada := "PU02_DB".p_auto,
                      pu02_man := "M_PU02_MAN",
                      pu02_man_scada := "PU02_DB".p_man,
                      pu02_mv := "PU02_DB".p_mv,
                      controller_cv := "LIC01_DB".CV,
                      controller_state => "CONTROLLER_STATE");
END_REGION

REGION Network 5
   RUNG wire#powerrail
      "Output Mapping"()
   END_RUNG
   // the same network as SCL:
   "Output Mapping"();
END_REGION
END_ORGANIZATION_BLOCK

ORGANIZATION_BLOCK "CyclicInterrupt(Regulator)"   // OB30, LAD, CyclicInterrupt
{ S7_Optimized_Access := 'TRUE' }
VERSION : 0.1
   VAR_INPUT
      Initial_Call : Bool;   // Initial call of this OB
      Event_Count : Int;   // Events discarded
   END_VAR
   VAR_TEMP
      compact_temp : Real;
   END_VAR
BEGIN

REGION Network 1
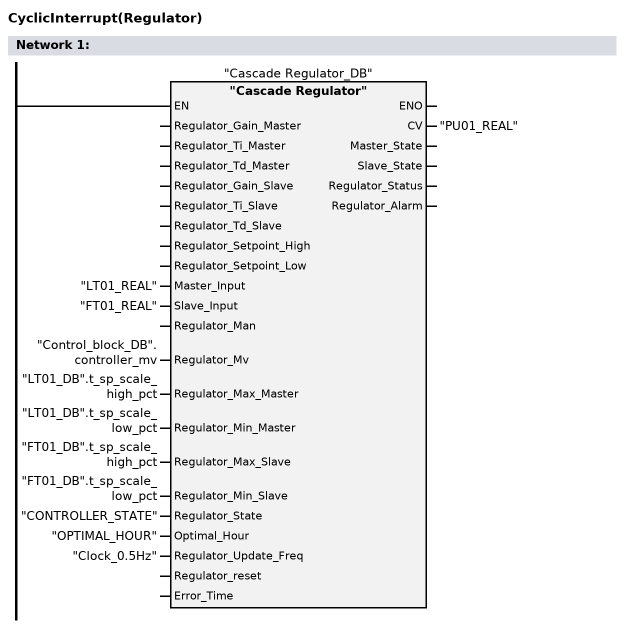
   RUNG wire#powerrail
      "Cascade Regulator_DB"(Regulator_Gain_Master :=, Regulator_Ti_Master :=, Regulator_Td_Master :=, Regulator_Gain_Slave :=, Regulator_Ti_Slave :=, Regulator_Td_Slave :=, Regulator_Setpoint_High :=, Regulator_Setpoint_Low :=, Master_Input := "LT01_REAL", Slave_Input := "FT01_REAL", Regulator_Man :=, Regulator_Mv := "Control_block_DB".controller_mv, Regulator_Max_Master := "LT01_DB".t_sp_scale_high_pct, Regulator_Min_Master := "LT01_DB".t_sp_scale_low_pct, Regulator_Max_Slave := "FT01_DB".t_sp_scale_high_pct, Regulator_Min_Slave := "FT01_DB".t_sp_scale_low_pct, Regulator_State := "CONTROLLER_STATE", Optimal_Hour := "OPTIMAL_HOUR", Regulator_Update_Freq := "Clock_0.5Hz", Regulator_reset :=, Error_Time :=, CV => "PU01_REAL", Master_State =>, Slave_State =>, Regulator_Status =>, Regulator_Alarm =>)
   END_RUNG
   // the same network as SCL:
   "Cascade Regulator_DB"(Master_Input := "LT01_REAL",   // "Cascade Regulator"
                          Slave_Input := "FT01_REAL",
                          Regulator_Mv := "Control_block_DB".controller_mv,
                          Regulator_Max_Master := "LT01_DB".t_sp_scale_high_pct,
                          Regulator_Min_Master := "LT01_DB".t_sp_scale_low_pct,
                          Regulator_Max_Slave := "FT01_DB".t_sp_scale_high_pct,
                          Regulator_Min_Slave := "FT01_DB".t_sp_scale_low_pct,
                          Regulator_State := "CONTROLLER_STATE",
                          Optimal_Hour := "OPTIMAL_HOUR",
                          Regulator_Update_Freq := "Clock_0.5Hz",
                          CV => "PU01_REAL");
END_REGION
END_ORGANIZATION_BLOCK

// folder: Modules

FUNCTION_BLOCK "Transmitter"   // FB2, LAD
{ S7_Optimized_Access := 'FALSE' }
VERSION : 0.1
   VAR_INPUT
      t_sp_hh_pct : Real := 3.8;   // transmitter setpoint high-high [%]
      t_sp_hh_sca : Real;   // transmitter setpoint high-high [m]
      t_sp_h_pct : Real := 3.5;   // transmitter setpoint high [%]
      t_sp_h_sca : Real;   // transmitter setpoint high [m]
      t_sp_l_pct : Real := 0.5;   // transmitter setpoint low [%]
      t_sp_l_sca : Real;   // transmitter setpoint low [m]
      t_sp_ll_pct : Real := 0.2;   // transmitter setpoint low-low [%]
      t_sp_ll_sca : Real;   // transmitter setpoint low-low [m]
      t_sp_scale_high_pct : Real := 4.0;   // transmitter setpoint scale high [%]
      t_sp_scale_high_sca : Real;   // transmitter setpoint scale high [m]
      t_sp_scale_low_pct : Real;   // transmitter setpoint scale low [%]
      t_sp_scale_low_sca : Real;   // transmitter setpoint scale low [%]
      t_hys : Int := 3;   // transmitter hysteresis [m]
      t_val : Int;   // transmitter value [Int]
      t_alarm_sec : Int := 5;   // the amount of time alarm signal has to be active to activate
      reset : Bool;
   END_VAR
   VAR_OUTPUT
      t_pv_pct : Real;   // transmitter process value
      t_pv_sca : Real;
   END_VAR
   VAR
      t_alarm_hh : Bool;
      t_alarm_h : Bool;
      t_alarm_l : Bool;
      t_alarm_ll : Bool;
      t_alarm_range : Bool;
      t_alarm : Bool;
      t_reset_scada : Bool;
      t_aw : Int;
      t_sp_hh_hys : Int;
      t_sp_h_hys : Int;
      t_sp_l_hys : Int;
      t_sp_ll_hys : Int;
      t_alarm_hys_temp : Int;
      t_alarm_hys : Time;
      t_alarm_time_temp : Int;
      t_alarm_time : Time;
   END_VAR
   VAR_TEMP
      t_temp : Real;
      t_pv_temp : Int;
   END_VAR
   VAR_TEMP   // added for the SCL form of the ladder/FBD networks
      _w1 : Bool;
   END_VAR
BEGIN

REGION Network 1
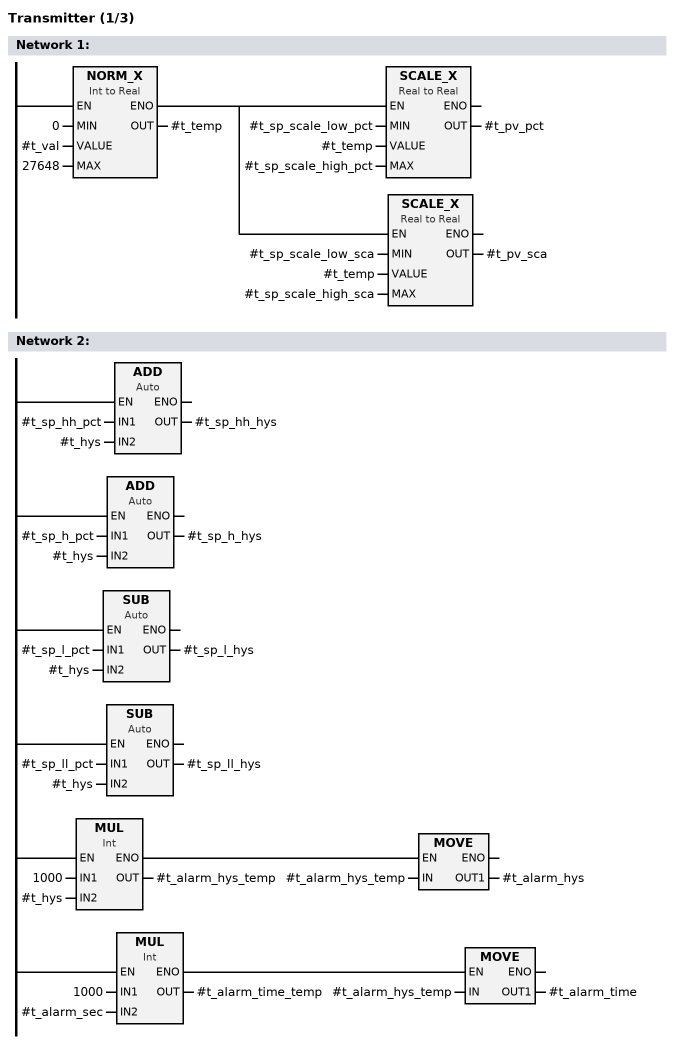
   RUNG wire#powerrail
      { S7_Templates := "[SrcType := Int, DestType := Real]"; S7_GenerateENO := "TRUE" } Normalize(min := 0, value := #t_val, max := 27648, out => #t_temp)
      wire#w1
      { S7_Templates := "[SrcType := Real, DestType := Real]"; S7_GenerateENO := "TRUE" } Scale(min := #t_sp_scale_low_pct, value := #t_temp, max := #t_sp_scale_high_pct, out => #t_pv_pct)
   END_RUNG
   RUNG wire#w1
      { S7_Templates := "[SrcType := Real, DestType := Real]"; S7_GenerateENO := "TRUE" } Scale(min := #t_sp_scale_low_sca, value := #t_temp, max := #t_sp_scale_high_sca, out => #t_pv_sca)
   END_RUNG
   // the same network as SCL:
   // ENO of a box is taken as its EN; it also drops when the box reports an error
   #t_temp := NORM_X(MIN := 0, VALUE := #t_val, MAX := 27648);
   #t_pv_pct := SCALE_X(MIN := #t_sp_scale_low_pct, VALUE := #t_temp, MAX := #t_sp_scale_high_pct);
   #t_pv_sca := SCALE_X(MIN := #t_sp_scale_low_sca, VALUE := #t_temp, MAX := #t_sp_scale_high_sca);
END_REGION

REGION Network 2
   RUNG wire#powerrail
      Add(in1 := #t_sp_hh_pct, in2 := #t_hys, out => #t_sp_hh_hys)
   END_RUNG
   RUNG wire#powerrail
      Add(in1 := #t_sp_h_pct, in2 := #t_hys, out => #t_sp_h_hys)
   END_RUNG
   RUNG wire#powerrail
      Sub(in1 := #t_sp_l_pct, in2 := #t_hys, out => #t_sp_l_hys)
   END_RUNG
   RUNG wire#powerrail
      Sub(in1 := #t_sp_ll_pct, in2 := #t_hys, out => #t_sp_ll_hys)
   END_RUNG
   RUNG wire#powerrail
      { S7_Templates := "SrcType := Int" } Mul(in1 := 1000, in2 := #t_hys, out => #t_alarm_hys_temp)
      Move(in := #t_alarm_hys_temp, out1 => #t_alarm_hys)
   END_RUNG
   RUNG wire#powerrail
      { S7_Templates := "SrcType := Int" } Mul(in1 := 1000, in2 := #t_alarm_sec, out => #t_alarm_time_temp)
      Move(in := #t_alarm_hys_temp, out1 => #t_alarm_time)
   END_RUNG
   // the same network as SCL:
   #t_sp_hh_hys := #t_sp_hh_pct + #t_hys;
   #t_sp_h_hys := #t_sp_h_pct + #t_hys;
   #t_sp_l_hys := #t_sp_l_pct - #t_hys;
   #t_sp_ll_hys := #t_sp_ll_pct - #t_hys;
   #t_alarm_hys_temp := 1000 * #t_hys;
   #t_alarm_hys := #t_alarm_hys_temp;
   #t_alarm_time_temp := 1000 * #t_alarm_sec;
   #t_alarm_time := #t_alarm_hys_temp;
END_REGION

REGION Network 3: transmitter alarm word
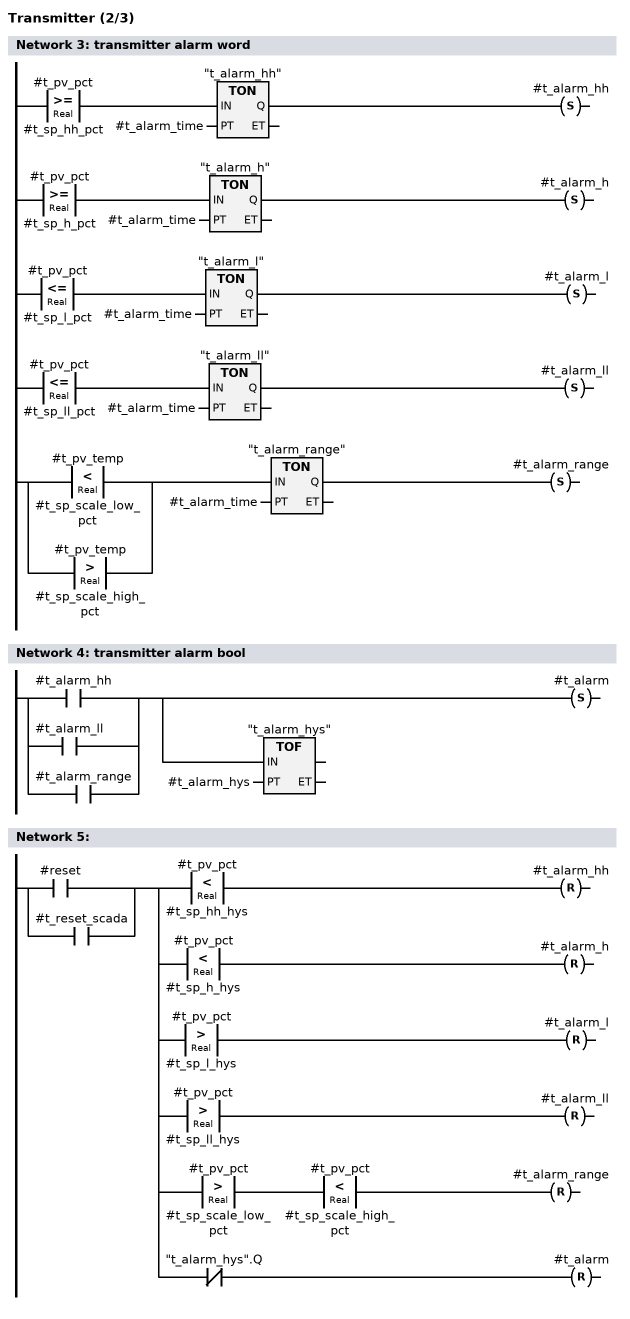
   "t_alarm_hh".TON(IN := #t_pv_pct >= #t_sp_hh_pct, PT := #t_alarm_time);
   IF "t_alarm_hh".Q THEN #t_alarm_hh := TRUE; END_IF;
   "t_alarm_h".TON(IN := #t_pv_pct >= #t_sp_h_pct, PT := #t_alarm_time);
   IF "t_alarm_h".Q THEN #t_alarm_h := TRUE; END_IF;
   "t_alarm_l".TON(IN := #t_pv_pct <= #t_sp_l_pct, PT := #t_alarm_time);
   IF "t_alarm_l".Q THEN #t_alarm_l := TRUE; END_IF;
   "t_alarm_ll".TON(IN := #t_pv_pct <= #t_sp_ll_pct, PT := #t_alarm_time);
   IF "t_alarm_ll".Q THEN #t_alarm_ll := TRUE; END_IF;
   "t_alarm_range".TON(IN := (#t_pv_temp < #t_sp_scale_low_pct) OR (#t_pv_temp > #t_sp_scale_high_pct),
                       PT := #t_alarm_time);
   IF "t_alarm_range".Q THEN #t_alarm_range := TRUE; END_IF;
END_REGION

REGION Network 4: transmitter alarm bool
   #_w1 := #t_alarm_hh OR #t_alarm_ll OR #t_alarm_range;
   IF #_w1 THEN #t_alarm := TRUE; END_IF;
   "t_alarm_hys".TOF(IN := #_w1, PT := #t_alarm_hys);
END_REGION

REGION Network 5
   RUNG wire#powerrail
      Contact( #reset )
      wire#w1
      { S7_Templates := "SrcType := Real" } LT_Contact(in1 := #t_pv_pct, in2 := #t_sp_hh_hys)
      R_Coil( #t_alarm_hh )
   END_RUNG
   RUNG wire#powerrail
      Contact( #t_reset_scada )
   END_RUNG wire#w1
   RUNG wire#w1
      { S7_Templates := "SrcType := Real" } LT_Contact(in1 := #t_pv_pct, in2 := #t_sp_h_hys)
      R_Coil( #t_alarm_h )
   END_RUNG
   RUNG wire#w1
      { S7_Templates := "SrcType := Real" } GT_Contact(in1 := #t_pv_pct, in2 := #t_sp_l_hys)
      R_Coil( #t_alarm_l )
   END_RUNG
   RUNG wire#w1
      { S7_Templates := "SrcType := Real" } GT_Contact(in1 := #t_pv_pct, in2 := #t_sp_ll_hys)
      R_Coil( #t_alarm_ll )
   END_RUNG
   RUNG wire#w1
      { S7_Templates := "SrcType := Real" } GT_Contact(in1 := #t_pv_pct, in2 := #t_sp_scale_low_pct)
      { S7_Templates := "SrcType := Real" } LT_Contact(in1 := #t_pv_pct, in2 := #t_sp_scale_high_pct)
      R_Coil( #t_alarm_range )
   END_RUNG
   RUNG wire#w1
      I_Contact( "t_alarm_hys".Q )
      R_Coil( #t_alarm )
   END_RUNG
   // the same network as SCL:
   #_w1 := #reset OR #t_reset_scada;
   IF #_w1 AND (#t_pv_pct < #t_sp_hh_hys) THEN #t_alarm_hh := FALSE; END_IF;
   IF #_w1 AND (#t_pv_pct < #t_sp_h_hys) THEN #t_alarm_h := FALSE; END_IF;
   IF #_w1 AND (#t_pv_pct > #t_sp_l_hys) THEN #t_alarm_l := FALSE; END_IF;
   IF #_w1 AND (#t_pv_pct > #t_sp_ll_hys) THEN #t_alarm_ll := FALSE; END_IF;
   IF #_w1 AND (#t_pv_pct > #t_sp_scale_low_pct) AND (#t_pv_pct < #t_sp_scale_high_pct) THEN
       #t_alarm_range := FALSE;
   END_IF;
   IF #_w1 AND NOT "t_alarm_hys".Q THEN #t_alarm := FALSE; END_IF;
END_REGION

REGION Network 6
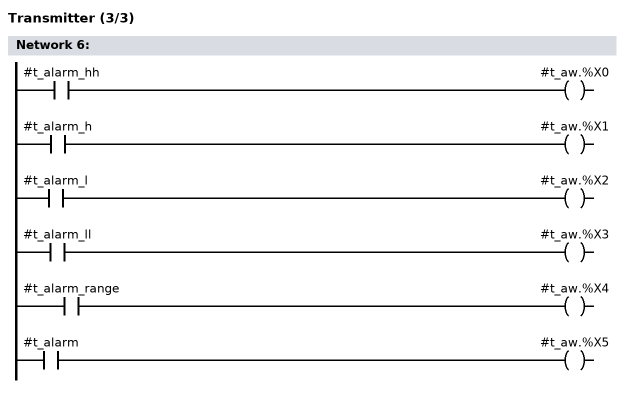
   RUNG wire#powerrail
      Contact( #t_alarm_hh )
      Coil( #t_aw.%X0 )
   END_RUNG
   RUNG wire#powerrail
      Contact( #t_alarm_h )
      Coil( #t_aw.%X1 )
   END_RUNG
   RUNG wire#powerrail
      Contact( #t_alarm_l )
      Coil( #t_aw.%X2 )
   END_RUNG
   RUNG wire#powerrail
      Contact( #t_alarm_ll )
      Coil( #t_aw.%X3 )
   END_RUNG
   RUNG wire#powerrail
      Contact( #t_alarm_range )
      Coil( #t_aw.%X4 )
   END_RUNG
   RUNG wire#powerrail
      Contact( #t_alarm )
      Coil( #t_aw.%X5 )
   END_RUNG
   // the same network as SCL:
   #t_aw.%X0 := #t_alarm_hh;
   #t_aw.%X1 := #t_alarm_h;
   #t_aw.%X2 := #t_alarm_l;
   #t_aw.%X3 := #t_alarm_ll;
   #t_aw.%X4 := #t_alarm_range;
   #t_aw.%X5 := #t_alarm;
END_REGION
END_FUNCTION_BLOCK

FUNCTION_BLOCK "Pump"   // FB3, LAD
{ S7_Optimized_Access := 'FALSE' }
VERSION : 0.1
   VAR_INPUT
      p_fwd : Bool;
      p_rev : Bool;
      p_fault_fv : Bool;
      p_fault_vfd : Bool;
      p_fault_tmp : Bool;
      p_fault_moi : Bool;
      p_reset : Bool;
      p_val : Real;
      p_scale_high : Int;
      p_scale_low : Int;
      p_hys : Int;
      p_alarm_sec : Int;
      p_auto_scada : Bool;
      p_man_scada : Bool;
      p_flow : Int;
      p_flow_ll : Int;
   END_VAR
   VAR_OUTPUT
      p_pv : Int;   // transmitter process value
      p_run : Bool;
      p_run_fwd : Bool;
      p_run_rev : Bool;
      p_fault : Bool;
      p_auto : Bool;
      p_man : Bool;
   END_VAR
   VAR_IN_OUT
      p_mv : Real;
   END_VAR
   VAR
      p_reset_scada : Bool;
      p_alarm_fv : Bool;
      p_alarm_vfd : Bool;
      p_alarm_tmp : Bool;
      p_alarm_moi : Bool;
      p_alarm_flow : Bool;
      p_alarm : Bool;
      p_aw : Int;
      p_alarm_time_temp : Int;
      p_alarm_time : Time;
   END_VAR
   VAR_TEMP
      p_temp : Real;
   END_VAR
   VAR_TEMP   // added for the SCL form of the ladder/FBD networks
      _w1 : Bool;
   END_VAR
BEGIN

REGION Network 1
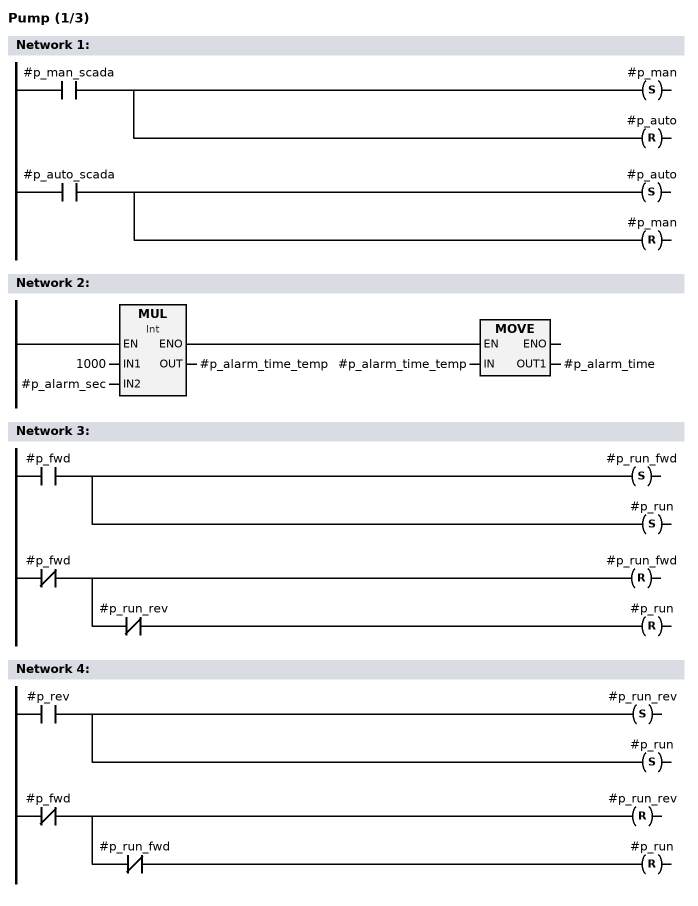
   RUNG wire#powerrail
      Contact( #p_man_scada )
      wire#w1
      S_Coil( #p_man )
   END_RUNG
   RUNG wire#w1
      R_Coil( #p_auto )
   END_RUNG
   RUNG wire#powerrail
      Contact( #p_auto_scada )
      wire#w2
      S_Coil( #p_auto )
   END_RUNG
   RUNG wire#w2
      R_Coil( #p_man )
   END_RUNG
   // the same network as SCL:
   IF #p_man_scada THEN
       #p_man := TRUE;
       #p_auto := FALSE;
   END_IF;
   IF #p_auto_scada THEN
       #p_auto := TRUE;
       #p_man := FALSE;
   END_IF;
END_REGION

REGION Network 2
   RUNG wire#powerrail
      { S7_Templates := "SrcType := Int" } Mul(in1 := 1000, in2 := #p_alarm_sec, out => #p_alarm_time_temp)
      Move(in := #p_alarm_time_temp, out1 => #p_alarm_time)
   END_RUNG
   // the same network as SCL:
   #p_alarm_time_temp := 1000 * #p_alarm_sec;
   #p_alarm_time := #p_alarm_time_temp;
END_REGION

REGION Network 3
   RUNG wire#powerrail
      Contact( #p_fwd )
      wire#w1
      S_Coil( #p_run_fwd )
   END_RUNG
   RUNG wire#w1
      S_Coil( #p_run )
   END_RUNG
   RUNG wire#powerrail
      I_Contact( #p_fwd )
      wire#w2
      R_Coil( #p_run_fwd )
   END_RUNG
   RUNG wire#w2
      I_Contact( #p_run_rev )
      R_Coil( #p_run )
   END_RUNG
   // the same network as SCL:
   IF #p_fwd THEN
       #p_run_fwd := TRUE;
       #p_run := TRUE;
   END_IF;
   IF NOT #p_fwd THEN #p_run_fwd := FALSE; END_IF;
   IF NOT #p_fwd AND NOT #p_run_rev THEN #p_run := FALSE; END_IF;
END_REGION

REGION Network 4
   RUNG wire#powerrail
      Contact( #p_rev )
      wire#w1
      S_Coil( #p_run_rev )
   END_RUNG
   RUNG wire#w1
      S_Coil( #p_run )
   END_RUNG
   RUNG wire#powerrail
      I_Contact( #p_fwd )
      wire#w2
      R_Coil( #p_run_rev )
   END_RUNG
   RUNG wire#w2
      I_Contact( #p_run_fwd )
      R_Coil( #p_run )
   END_RUNG
   // the same network as SCL:
   IF #p_rev THEN
       #p_run_rev := TRUE;
       #p_run := TRUE;
   END_IF;
   IF NOT #p_fwd THEN #p_run_rev := FALSE; END_IF;
   IF NOT #p_fwd AND NOT #p_run_fwd THEN #p_run := FALSE; END_IF;
END_REGION

REGION Network 5
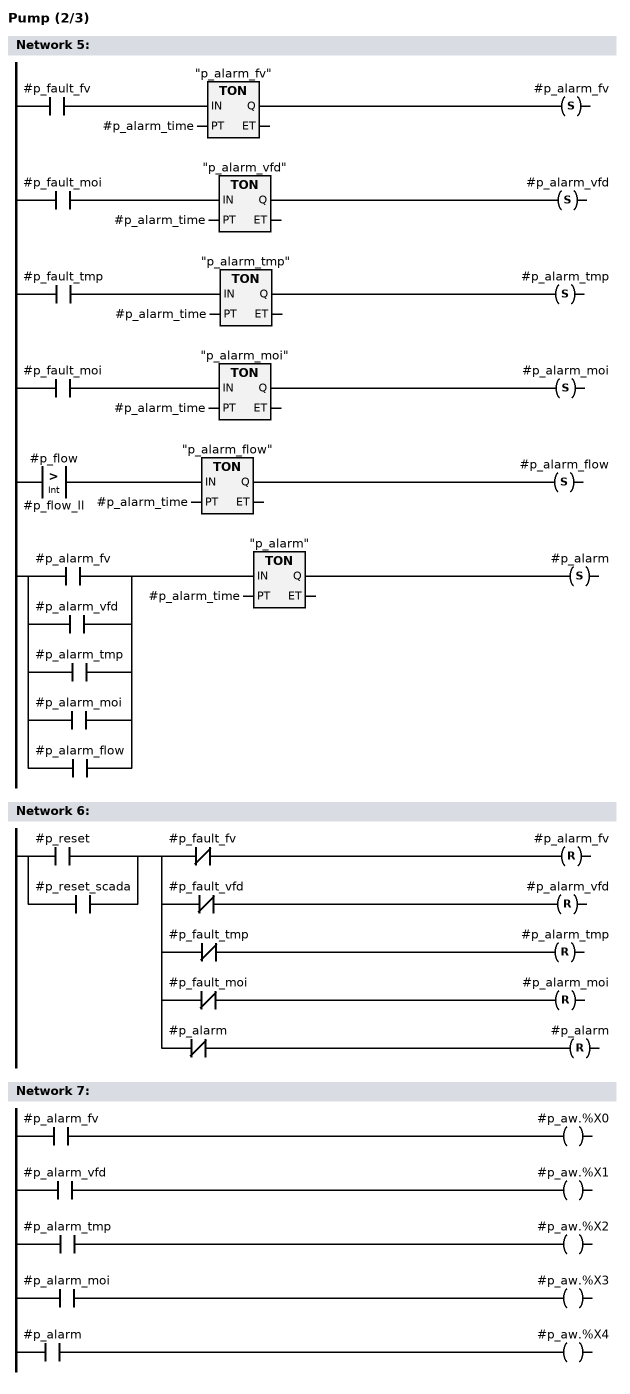
   "p_alarm_fv".TON(IN := #p_fault_fv, PT := #p_alarm_time);
   IF "p_alarm_fv".Q THEN #p_alarm_fv := TRUE; END_IF;
   "p_alarm_vfd".TON(IN := #p_fault_moi, PT := #p_alarm_time);
   IF "p_alarm_vfd".Q THEN #p_alarm_vfd := TRUE; END_IF;
   "p_alarm_tmp".TON(IN := #p_fault_tmp, PT := #p_alarm_time);
   IF "p_alarm_tmp".Q THEN #p_alarm_tmp := TRUE; END_IF;
   "p_alarm_moi".TON(IN := #p_fault_moi, PT := #p_alarm_time);
   IF "p_alarm_moi".Q THEN #p_alarm_moi := TRUE; END_IF;
   "p_alarm_flow".TON(IN := #p_flow > #p_flow_ll, PT := #p_alarm_time);
   IF "p_alarm_flow".Q THEN #p_alarm_flow := TRUE; END_IF;
   "p_alarm".TON(IN := #p_alarm_fv OR #p_alarm_vfd OR #p_alarm_tmp OR #p_alarm_moi OR #p_alarm_flow,
                 PT := #p_alarm_time);
   IF "p_alarm".Q THEN #p_alarm := TRUE; END_IF;
END_REGION

REGION Network 6
   RUNG wire#powerrail
      Contact( #p_reset )
      wire#w1
      I_Contact( #p_fault_fv )
      R_Coil( #p_alarm_fv )
   END_RUNG
   RUNG wire#powerrail
      Contact( #p_reset_scada )
   END_RUNG wire#w1
   RUNG wire#w1
      I_Contact( #p_fault_vfd )
      R_Coil( #p_alarm_vfd )
   END_RUNG
   RUNG wire#w1
      I_Contact( #p_fault_tmp )
      R_Coil( #p_alarm_tmp )
   END_RUNG
   RUNG wire#w1
      I_Contact( #p_fault_moi )
      R_Coil( #p_alarm_moi )
   END_RUNG
   RUNG wire#w1
      I_Contact( #p_alarm )
      R_Coil( #p_alarm )
   END_RUNG
   // the same network as SCL:
   #_w1 := #p_reset OR #p_reset_scada;
   IF #_w1 AND NOT #p_fault_fv THEN #p_alarm_fv := FALSE; END_IF;
   IF #_w1 AND NOT #p_fault_vfd THEN #p_alarm_vfd := FALSE; END_IF;
   IF #_w1 AND NOT #p_fault_tmp THEN #p_alarm_tmp := FALSE; END_IF;
   IF #_w1 AND NOT #p_fault_moi THEN #p_alarm_moi := FALSE; END_IF;
   IF #_w1 AND NOT #p_alarm THEN #p_alarm := FALSE; END_IF;
END_REGION

REGION Network 7
   RUNG wire#powerrail
      Contact( #p_alarm_fv )
      Coil( #p_aw.%X0 )
   END_RUNG
   RUNG wire#powerrail
      Contact( #p_alarm_vfd )
      Coil( #p_aw.%X1 )
   END_RUNG
   RUNG wire#powerrail
      Contact( #p_alarm_tmp )
      Coil( #p_aw.%X2 )
   END_RUNG
   RUNG wire#powerrail
      Contact( #p_alarm_moi )
      Coil( #p_aw.%X3 )
   END_RUNG
   RUNG wire#powerrail
      Contact( #p_alarm )
      Coil( #p_aw.%X4 )
   END_RUNG
   // the same network as SCL:
   #p_aw.%X0 := #p_alarm_fv;
   #p_aw.%X1 := #p_alarm_vfd;
   #p_aw.%X2 := #p_alarm_tmp;
   #p_aw.%X3 := #p_alarm_moi;
   #p_aw.%X4 := #p_alarm;
END_REGION

REGION Network 8
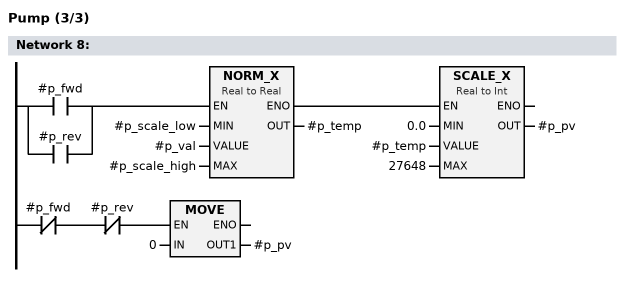
   RUNG wire#powerrail
      Contact( #p_fwd )
      wire#w1
      { S7_Templates := "[SrcType := Real, DestType := Real]"; S7_GenerateENO := "TRUE" } Normalize(min := #p_scale_low, value := #p_val, max := #p_scale_high, out => #p_temp)
      { S7_Templates := "[SrcType := Real, DestType := Int]"; S7_GenerateENO := "TRUE" } Scale(min := 0.0, value := #p_temp, max := 27648, out => #p_pv)
   END_RUNG
   RUNG wire#powerrail
      Contact( #p_rev )
   END_RUNG wire#w1
   RUNG wire#powerrail
      I_Contact( #p_fwd )
      I_Contact( #p_rev )
      Move(in := 0, out1 => #p_pv)
   END_RUNG
   // the same network as SCL:
   // ENO of a box is taken as its EN; it also drops when the box reports an error
   IF #p_fwd OR #p_rev THEN
       #p_temp := NORM_X(MIN := #p_scale_low, VALUE := #p_val, MAX := #p_scale_high);
       #p_pv := SCALE_X(MIN := 0.0, VALUE := #p_temp, MAX := 27648);
   END_IF;
   IF NOT #p_fwd AND NOT #p_rev THEN #p_pv := 0; END_IF;
END_REGION
END_FUNCTION_BLOCK

FUNCTION_BLOCK "Cascade Regulator"   // FB7, LAD
{ S7_Optimized_Access := 'FALSE' }
VERSION : 0.1
   VAR_INPUT
      Regulator_Gain_Primary : Real := 125.0;
      Regulator_Ti_Primary : Real := 2.72;
      Regulator_Td_Primary : Real;
      Regulator_Gain_Secondary : Real := 0.2;
      Regulator_Ti_Secondary : Real := 3.0;
      Regulator_Td_Secondary : Real;
      Regulator_Setpoint_High : Real := 75.0;
      Regulator_Setpoint_Low : Real := 50.0;
      Primary_Input : Real;
      Secondary_Input : Real;
      Regulator_Man : Bool;
      Regulator_Mv : Real;
      Regulator_Max_Primary : Real := 100.0;
      Regulator_Min_Primary : Real := 0.0;
      Regulator_Max_Secondary : Real := 100.0;
      Regulator_Min_Secondary : Real;
      Regulator_State : Int;
      Optimal_Hour : Bool;
      Regulator_Update_Freq : Bool;
      Regulator_reset : Bool;
      Error_Time : Int := 1;   // Amount of time it takes for an alarm to get activated [S]
   END_VAR
   VAR_OUTPUT
      CV : Real;
      Primary_State : Int;
      Secondary_State : Int;
      Regulator_Status : Int;
      Regulator_Alarm : Bool;
   END_VAR
   VAR
      Regulator_Setpoint : Real;
      Regulator_Automatic : Bool;
      Regulator_Manual : Bool;
      "Input Error" : Bool;
      "Tuning Error" : Bool;
      "Setpoint Error" : Bool;
      "ManualValue Error" : Bool;
      "General Error" : Bool;
      "Regulator Error" : Bool;
      reset_controller_scada : Bool;   // Resets the controllers faults from scada
      reset_controller_memory : Bool;   // Resets the controllers controller every stop
      Regulator_Stopped : Bool;
      Alarm_Time : Time;
      Error_Time_Temp : Int;
      CV_unmod : Real;
      CV_min : Bool;
      trig_0 : Bool;
      trig_1 : Bool;
      trig_2 : Bool;
      trig_3 : Bool;
   END_VAR
   VAR_TEMP
      compact_temp : Real;
   END_VAR
   VAR_TEMP   // added for the SCL form of the ladder/FBD networks
      _w1 : Bool;
      _w2 : Bool;
      _w3 : Bool;
      _w4 : Bool;
   END_VAR
BEGIN

REGION Network 1: PID Values
   // Sets the PID values for the regulator
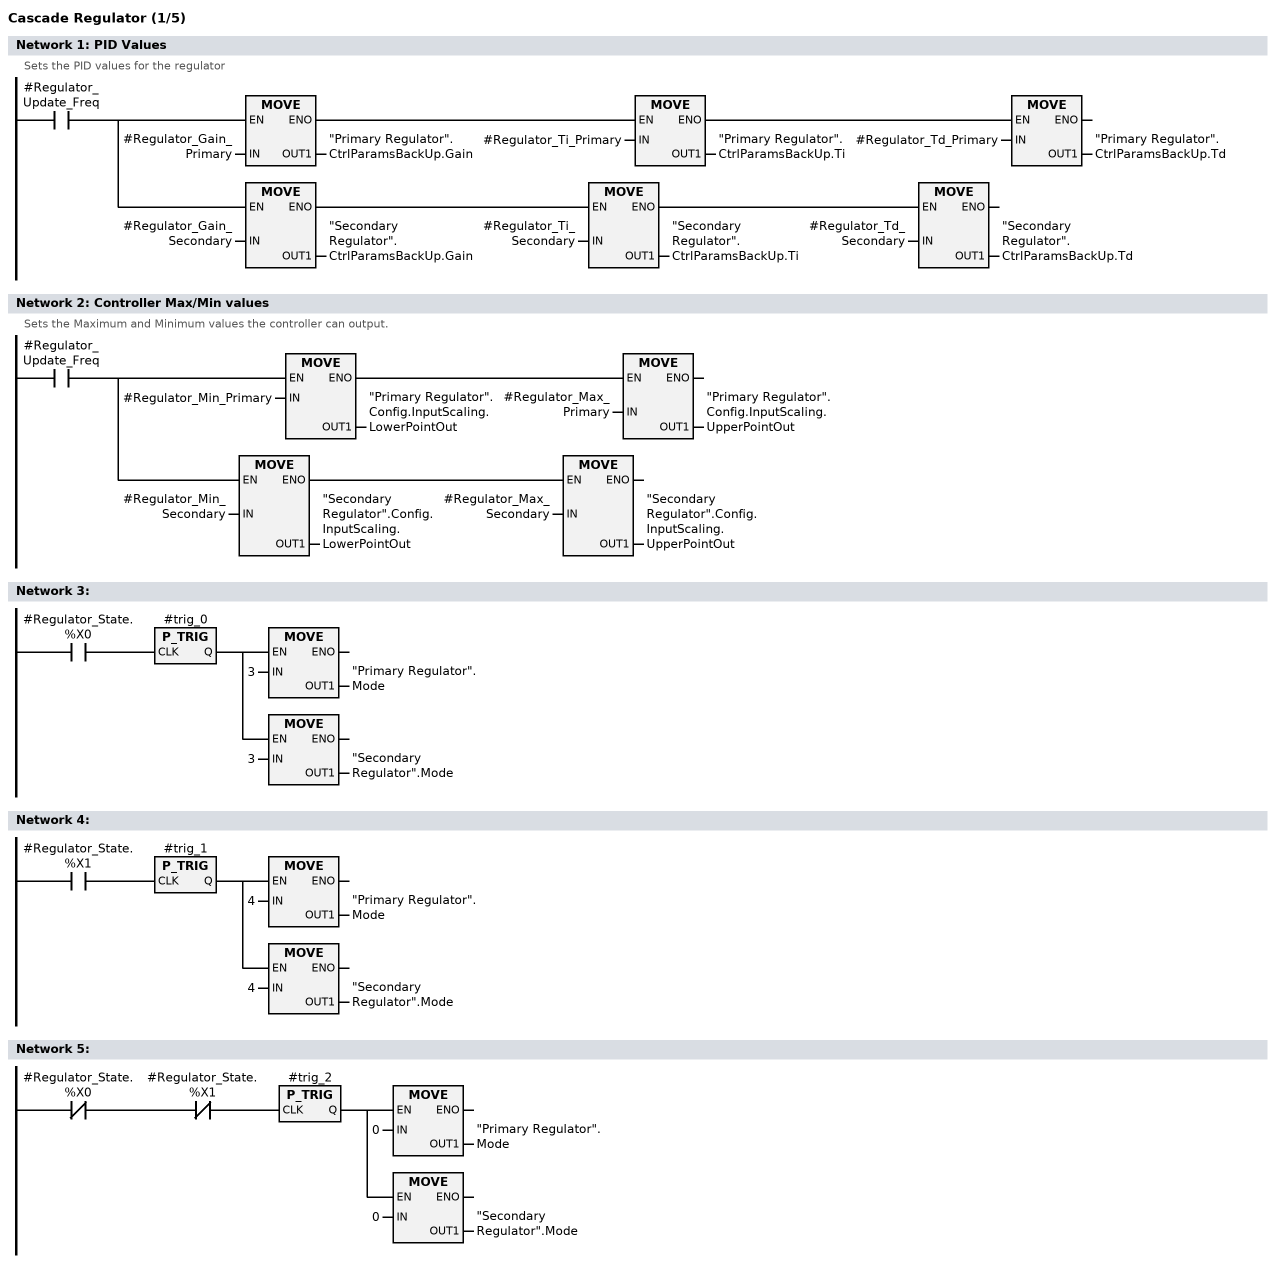
   RUNG wire#powerrail
      Contact( #Regulator_Update_Freq )
      wire#w1
      Move(in := #Regulator_Gain_Primary, out1 => "Primary Regulator".CtrlParamsBackUp.Gain)
      Move(in := #Regulator_Ti_Primary, out1 => "Primary Regulator".CtrlParamsBackUp.Ti)
      Move(in := #Regulator_Td_Primary, out1 => "Primary Regulator".CtrlParamsBackUp.Td)
   END_RUNG
   RUNG wire#w1
      Move(in := #Regulator_Gain_Secondary, out1 => "Secondary Regulator".CtrlParamsBackUp.Gain)
      Move(in := #Regulator_Ti_Secondary, out1 => "Secondary Regulator".CtrlParamsBackUp.Ti)
      Move(in := #Regulator_Td_Secondary, out1 => "Secondary Regulator".CtrlParamsBackUp.Td)
   END_RUNG
   // the same network as SCL:
   IF #Regulator_Update_Freq THEN
       "Primary Regulator".CtrlParamsBackUp.Gain := #Regulator_Gain_Primary;
       "Primary Regulator".CtrlParamsBackUp.Ti := #Regulator_Ti_Primary;
       "Primary Regulator".CtrlParamsBackUp.Td := #Regulator_Td_Primary;
       "Secondary Regulator".CtrlParamsBackUp.Gain := #Regulator_Gain_Secondary;
       "Secondary Regulator".CtrlParamsBackUp.Ti := #Regulator_Ti_Secondary;
       "Secondary Regulator".CtrlParamsBackUp.Td := #Regulator_Td_Secondary;
   END_IF;
END_REGION

REGION Network 2: Controller Max/Min values
   // Sets the Maximum and Minimum values the controller can output.
   RUNG wire#powerrail
      Contact( #Regulator_Update_Freq )
      wire#w1
      Move(in := #Regulator_Min_Primary, out1 => "Primary Regulator".Config.InputScaling.LowerPointOut)
      Move(in := #Regulator_Max_Primary, out1 => "Primary Regulator".Config.InputScaling.UpperPointOut)
   END_RUNG
   RUNG wire#w1
      Move(in := #Regulator_Min_Secondary, out1 => "Secondary Regulator".Config.InputScaling.LowerPointOut)
      Move(in := #Regulator_Max_Secondary, out1 => "Secondary Regulator".Config.InputScaling.UpperPointOut)
   END_RUNG
   // the same network as SCL:
   IF #Regulator_Update_Freq THEN
       "Primary Regulator".Config.InputScaling.LowerPointOut := #Regulator_Min_Primary;
       "Primary Regulator".Config.InputScaling.UpperPointOut := #Regulator_Max_Primary;
       "Secondary Regulator".Config.InputScaling.LowerPointOut := #Regulator_Min_Secondary;
       "Secondary Regulator".Config.InputScaling.UpperPointOut := #Regulator_Max_Secondary;
   END_IF;
END_REGION

REGION Network 3
   RUNG wire#powerrail
      Contact( #Regulator_State.%X0 )
      P_Trig( #trig_0 )
      wire#w1
      Move(in := 3, out1 => "Primary Regulator".Mode)
   END_RUNG
   RUNG wire#w1
      Move(in := 3, out1 => "Secondary Regulator".Mode)
   END_RUNG
   // the same network as SCL:
   #_w1 := #Regulator_State.%X0 AND NOT #trig_0;   // rising edge
   #trig_0 := #Regulator_State.%X0;
   IF #_w1 THEN
       "Primary Regulator".Mode := 3;
       "Secondary Regulator".Mode := 3;
   END_IF;
END_REGION

REGION Network 4
   RUNG wire#powerrail
      Contact( #Regulator_State.%X1 )
      P_Trig( #trig_1 )
      wire#w1
      Move(in := 4, out1 => "Primary Regulator".Mode)
   END_RUNG
   RUNG wire#w1
      Move(in := 4, out1 => "Secondary Regulator".Mode)
   END_RUNG
   // the same network as SCL:
   #_w1 := #Regulator_State.%X1 AND NOT #trig_1;   // rising edge
   #trig_1 := #Regulator_State.%X1;
   IF #_w1 THEN
       "Primary Regulator".Mode := 4;
       "Secondary Regulator".Mode := 4;
   END_IF;
END_REGION

REGION Network 5
   RUNG wire#powerrail
      I_Contact( #Regulator_State.%X0 )
      I_Contact( #Regulator_State.%X1 )
      P_Trig( #trig_2 )
      wire#w1
      Move(in := 0, out1 => "Primary Regulator".Mode)
   END_RUNG
   RUNG wire#w1
      Move(in := 0, out1 => "Secondary Regulator".Mode)
   END_RUNG
   // the same network as SCL:
   #_w1 := NOT #Regulator_State.%X0 AND NOT #Regulator_State.%X1;
   #_w2 := #_w1 AND NOT #trig_2;   // rising edge
   #trig_2 := #_w1;
   IF #_w2 THEN
       "Primary Regulator".Mode := 0;
       "Secondary Regulator".Mode := 0;
   END_IF;
END_REGION

REGION Network 6: Reset Controller
   // Resets the controller everytime the controller gets stopped, so the output dosent stay the same when the controller starts after being stopped.
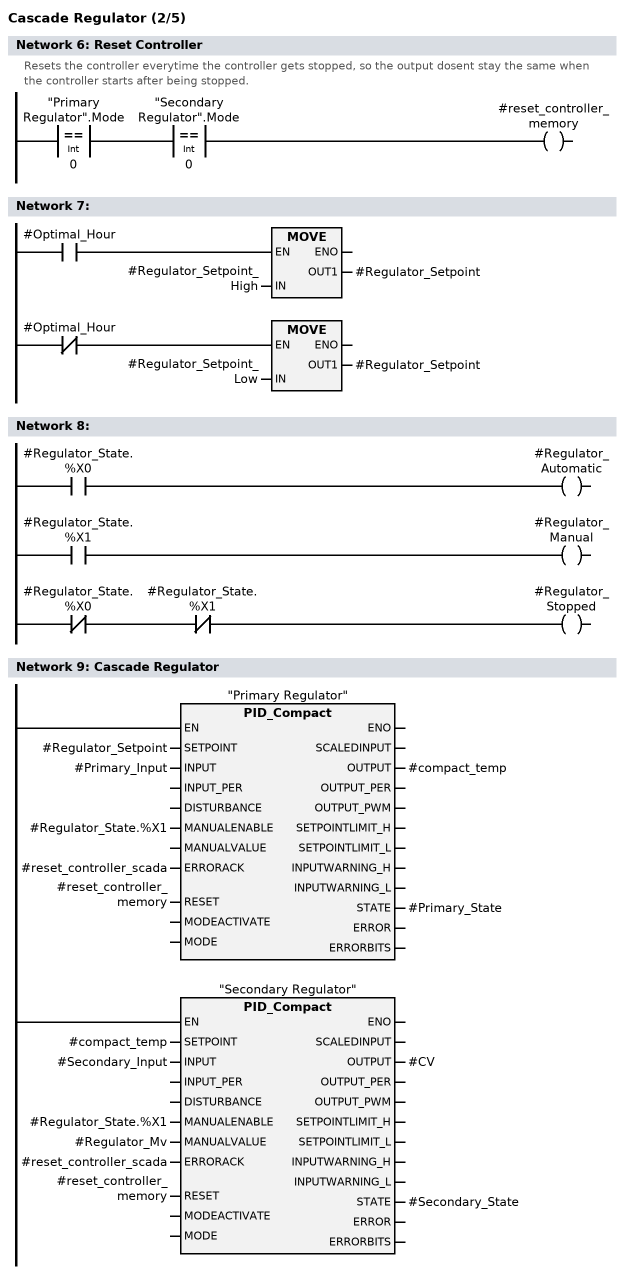
   RUNG wire#powerrail
      { S7_Templates := "SrcType := Int" } EQ_Contact(in1 := "Primary Regulator".Mode, in2 := 0)
      { S7_Templates := "SrcType := Int" } EQ_Contact(in1 := "Secondary Regulator".Mode, in2 := 0)
      Coil( #reset_controller_memory )
   END_RUNG
   // the same network as SCL:
   #reset_controller_memory := ("Primary Regulator".Mode = 0) AND ("Secondary Regulator".Mode = 0);
END_REGION

REGION Network 7
   RUNG wire#powerrail
      Contact( #Optimal_Hour )
      Move(in := #Regulator_Setpoint_High, out1 => #Regulator_Setpoint)
   END_RUNG
   RUNG wire#powerrail
      I_Contact( #Optimal_Hour )
      Move(in := #Regulator_Setpoint_Low, out1 => #Regulator_Setpoint)
   END_RUNG
   // the same network as SCL:
   IF #Optimal_Hour THEN #Regulator_Setpoint := #Regulator_Setpoint_High; END_IF;
   IF NOT #Optimal_Hour THEN #Regulator_Setpoint := #Regulator_Setpoint_Low; END_IF;
END_REGION

REGION Network 8
   RUNG wire#powerrail
      Contact( #Regulator_State.%X0 )
      Coil( #Regulator_Automatic )
   END_RUNG
   RUNG wire#powerrail
      Contact( #Regulator_State.%X1 )
      Coil( #Regulator_Manual )
   END_RUNG
   RUNG wire#powerrail
      I_Contact( #Regulator_State.%X0 )
      I_Contact( #Regulator_State.%X1 )
      Coil( #Regulator_Stopped )
   END_RUNG
   // the same network as SCL:
   #Regulator_Automatic := #Regulator_State.%X0;
   #Regulator_Manual := #Regulator_State.%X1;
   #Regulator_Stopped := NOT #Regulator_State.%X0 AND NOT #Regulator_State.%X1;
END_REGION

REGION Network 9: Cascade Regulator
   "Primary Regulator"(Setpoint := #Regulator_Setpoint,   // PID_Compact
                       Input := #Primary_Input,
                       ManualEnable := #Regulator_State.%X1,
                       ErrorAck := #reset_controller_scada,
                       Reset := #reset_controller_memory,
                       Output => #compact_temp,
                       State => #Primary_State);
   "Secondary Regulator"(Setpoint := #compact_temp,   // PID_Compact
                         Input := #Secondary_Input,
                         ManualEnable := #Regulator_State.%X1,
                         ManualValue := #Regulator_Mv,
                         ErrorAck := #reset_controller_scada,
                         Reset := #reset_controller_memory,
                         Output => #CV,
                         State => #Secondary_State);
END_REGION

REGION Network 10
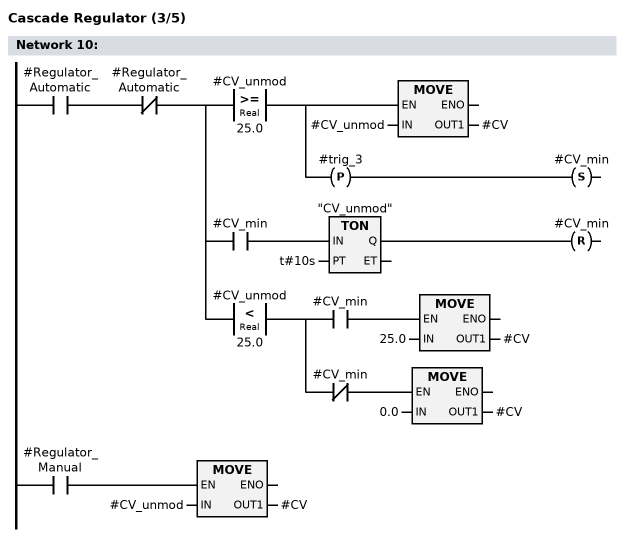
   #_w1 := #Regulator_Automatic AND NOT #Regulator_Automatic;
   #_w2 := #_w1 AND (#CV_unmod >= 25.0);
   IF #_w2 THEN #CV := #CV_unmod; END_IF;
   #_w3 := #_w2 AND NOT #trig_3;   // rising edge
   #trig_3 := #_w2;
   IF #_w3 THEN #CV_min := TRUE; END_IF;
   "CV_unmod".TON(IN := #_w1 AND #CV_min, PT := t#10s);
   IF "CV_unmod".Q THEN #CV_min := FALSE; END_IF;
   #_w4 := #_w1 AND (#CV_unmod < 25.0);
   IF #_w4 AND #CV_min THEN #CV := 25.0; END_IF;
   IF #_w4 AND NOT #CV_min THEN #CV := 0.0; END_IF;
   IF #Regulator_Manual THEN #CV := #CV_unmod; END_IF;
END_REGION

REGION Network 11: Controller Status
   // Sets different bits in the alarm word and forwards it.
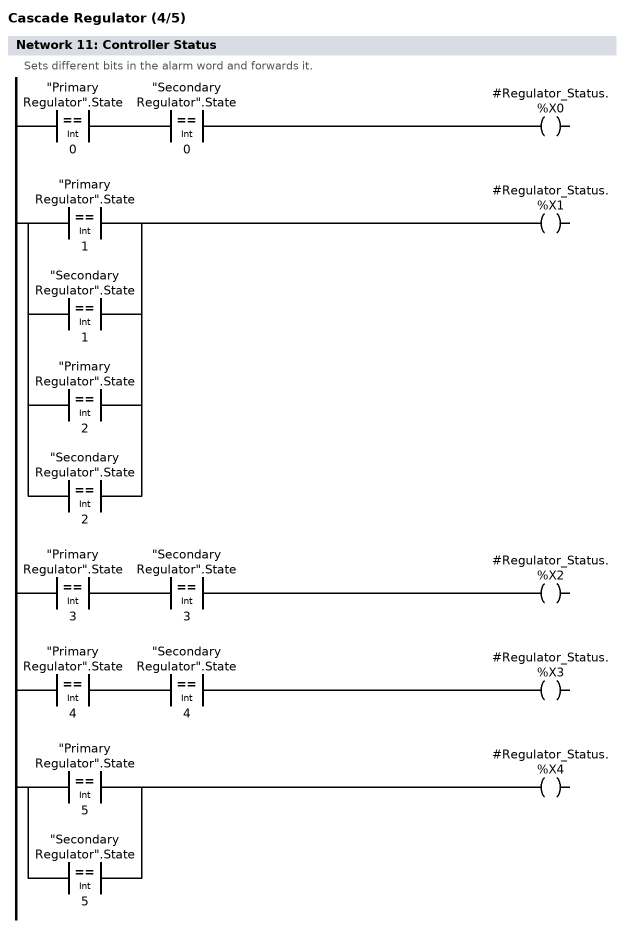
   RUNG wire#powerrail
      { S7_Templates := "SrcType := Int" } EQ_Contact(in1 := "Primary Regulator".State, in2 := 0)
      { S7_Templates := "SrcType := Int" } EQ_Contact(in1 := "Secondary Regulator".State, in2 := 0)
      Coil( #Regulator_Status.%X0 )
   END_RUNG
   RUNG wire#powerrail
      { S7_Templates := "SrcType := Int" } EQ_Contact(in1 := "Primary Regulator".State, in2 := 1)
      wire#w1
      Coil( #Regulator_Status.%X1 )
   END_RUNG
   RUNG wire#powerrail
      { S7_Templates := "SrcType := Int" } EQ_Contact(in1 := "Secondary Regulator".State, in2 := 1)
   END_RUNG wire#w1
   RUNG wire#powerrail
      { S7_Templates := "SrcType := Int" } EQ_Contact(in1 := "Primary Regulator".State, in2 := 2)
   END_RUNG wire#w1
   RUNG wire#powerrail
      { S7_Templates := "SrcType := Int" } EQ_Contact(in1 := "Secondary Regulator".State, in2 := 2)
   END_RUNG wire#w1
   RUNG wire#powerrail
      { S7_Templates := "SrcType := Int" } EQ_Contact(in1 := "Primary Regulator".State, in2 := 3)
      { S7_Templates := "SrcType := Int" } EQ_Contact(in1 := "Secondary Regulator".State, in2 := 3)
      Coil( #Regulator_Status.%X2 )
   END_RUNG
   RUNG wire#powerrail
      { S7_Templates := "SrcType := Int" } EQ_Contact(in1 := "Primary Regulator".State, in2 := 4)
      { S7_Templates := "SrcType := Int" } EQ_Contact(in1 := "Secondary Regulator".State, in2 := 4)
      Coil( #Regulator_Status.%X3 )
   END_RUNG
   RUNG wire#powerrail
      { S7_Templates := "SrcType := Int" } EQ_Contact(in1 := "Primary Regulator".State, in2 := 5)
      wire#w2
      Coil( #Regulator_Status.%X4 )
   END_RUNG
   RUNG wire#powerrail
      { S7_Templates := "SrcType := Int" } EQ_Contact(in1 := "Secondary Regulator".State, in2 := 5)
   END_RUNG wire#w2
   // the same network as SCL:
   #Regulator_Status.%X0 := ("Primary Regulator".State = 0) AND ("Secondary Regulator".State = 0);
   #Regulator_Status.%X1 := ("Primary Regulator".State = 1) OR ("Secondary Regulator".State = 1) OR ("Primary Regulator".State = 2) OR ("Secondary Regulator".State = 2);
   #Regulator_Status.%X2 := ("Primary Regulator".State = 3) AND ("Secondary Regulator".State = 3);
   #Regulator_Status.%X3 := ("Primary Regulator".State = 4) AND ("Secondary Regulator".State = 4);
   #Regulator_Status.%X4 := ("Primary Regulator".State = 5) OR ("Secondary Regulator".State = 5);
END_REGION

REGION Network 12: Controller Error
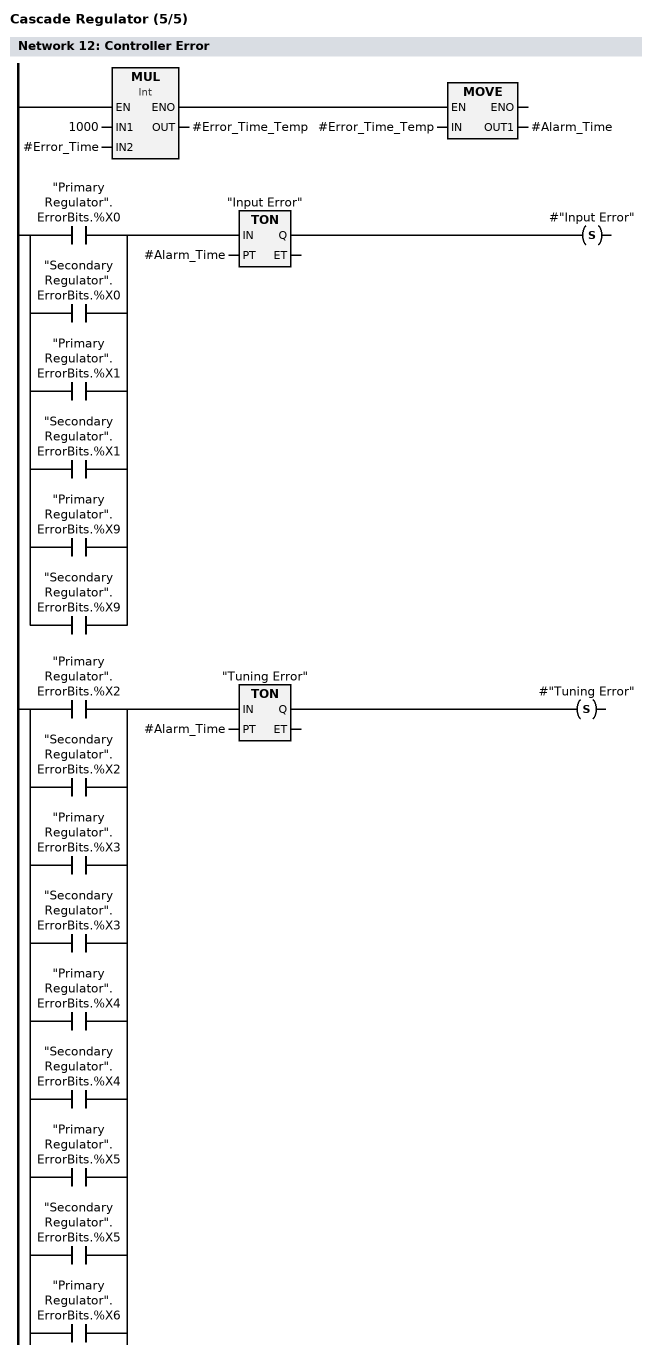
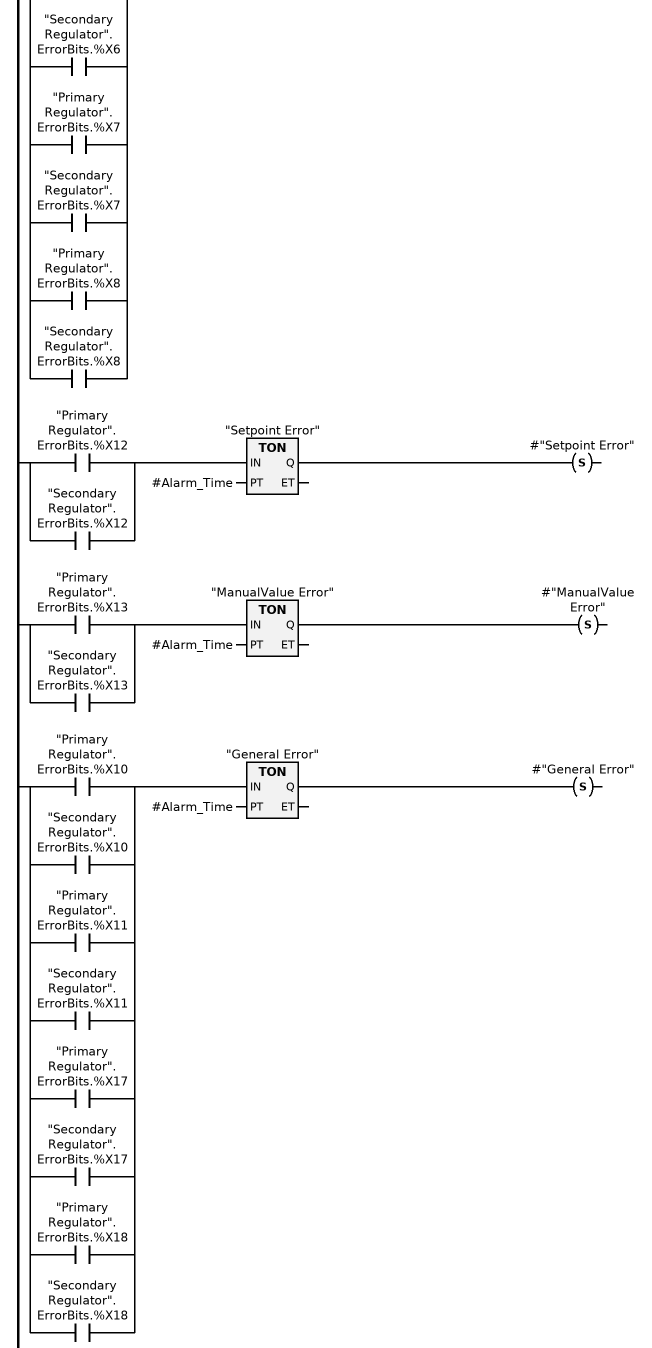
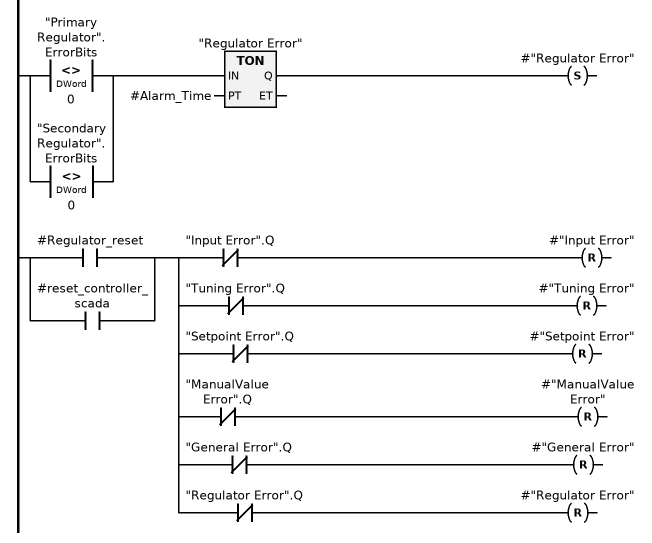
   #Error_Time_Temp := 1000 * #Error_Time;
   #Alarm_Time := #Error_Time_Temp;
   "Input Error".TON(IN := "Primary Regulator".ErrorBits.%X0 OR "Secondary Regulator".ErrorBits.%X0 OR "Primary Regulator".ErrorBits.%X1 OR "Secondary Regulator".ErrorBits.%X1 OR "Primary Regulator".ErrorBits.%X9 OR "Secondary Regulator".ErrorBits.%X9,
                     PT := #Alarm_Time);
   IF "Input Error".Q THEN #"Input Error" := TRUE; END_IF;
   "Tuning Error".TON(IN := "Primary Regulator".ErrorBits.%X2 OR "Secondary Regulator".ErrorBits.%X2 OR "Primary Regulator".ErrorBits.%X3 OR "Secondary Regulator".ErrorBits.%X3 OR "Primary Regulator".ErrorBits.%X4 OR "Secondary Regulator".ErrorBits.%X4 OR "Primary Regulator".ErrorBits.%X5 OR "Secondary Regulator".ErrorBits.%X5 OR "Primary Regulator".ErrorBits.%X6 OR "Secondary Regulator".ErrorBits.%X6 OR "Primary Regulator".ErrorBits.%X7 OR "Secondary Regulator".ErrorBits.%X7 OR "Primary Regulator".ErrorBits.%X8 OR "Secondary Regulator".ErrorBits.%X8,
                      PT := #Alarm_Time);
   IF "Tuning Error".Q THEN #"Tuning Error" := TRUE; END_IF;
   "Setpoint Error".TON(IN := "Primary Regulator".ErrorBits.%X12 OR "Secondary Regulator".ErrorBits.%X12,
                        PT := #Alarm_Time);
   IF "Setpoint Error".Q THEN #"Setpoint Error" := TRUE; END_IF;
   "ManualValue Error".TON(IN := "Primary Regulator".ErrorBits.%X13 OR "Secondary Regulator".ErrorBits.%X13,
                           PT := #Alarm_Time);
   IF "ManualValue Error".Q THEN #"ManualValue Error" := TRUE; END_IF;
   "General Error".TON(IN := "Primary Regulator".ErrorBits.%X10 OR "Secondary Regulator".ErrorBits.%X10 OR "Primary Regulator".ErrorBits.%X11 OR "Secondary Regulator".ErrorBits.%X11 OR "Primary Regulator".ErrorBits.%X17 OR "Secondary Regulator".ErrorBits.%X17 OR "Primary Regulator".ErrorBits.%X18 OR "Secondary Regulator".ErrorBits.%X18,
                       PT := #Alarm_Time);
   IF "General Error".Q THEN #"General Error" := TRUE; END_IF;
   "Regulator Error".TON(IN := ("Primary Regulator".ErrorBits <> 0) OR ("Secondary Regulator".ErrorBits <> 0),
                         PT := #Alarm_Time);
   IF "Regulator Error".Q THEN #"Regulator Error" := TRUE; END_IF;
   #_w1 := #Regulator_reset OR #reset_controller_scada;
   IF #_w1 AND NOT "Input Error".Q THEN #"Input Error" := FALSE; END_IF;
   IF #_w1 AND NOT "Tuning Error".Q THEN #"Tuning Error" := FALSE; END_IF;
   IF #_w1 AND NOT "Setpoint Error".Q THEN #"Setpoint Error" := FALSE; END_IF;
   IF #_w1 AND NOT "ManualValue Error".Q THEN #"ManualValue Error" := FALSE; END_IF;
   IF #_w1 AND NOT "General Error".Q THEN #"General Error" := FALSE; END_IF;
   IF #_w1 AND NOT "Regulator Error".Q THEN #"Regulator Error" := FALSE; END_IF;
END_REGION
END_FUNCTION_BLOCK

FUNCTION "Check optimal hour" : Void   // FC2, LAD
{ S7_Optimized_Access := 'TRUE' }
VERSION : 0.1
   VAR_INPUT
      electricitycost_dint : DInt;
   END_VAR
   VAR_OUTPUT
      optimal_hour : Bool;
   END_VAR
   VAR_TEMP
      date_and_time : Date_And_Time;
      "date_and_time_fault-code" : Int;
      time_of_day : Time_Of_Day;
   END_VAR
BEGIN

REGION Network 1: Convert Date_And_Time to Time_Of_Day
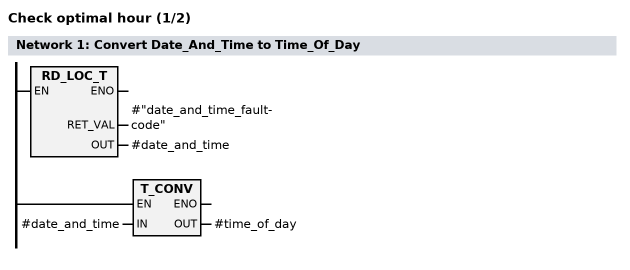
   #"date_and_time_fault-code" := RD_LOC_T(OUT => #date_and_time);
   #time_of_day := T_CONV(IN := #date_and_time);
END_REGION

REGION Network 2: Check if it's currently an optimal hour
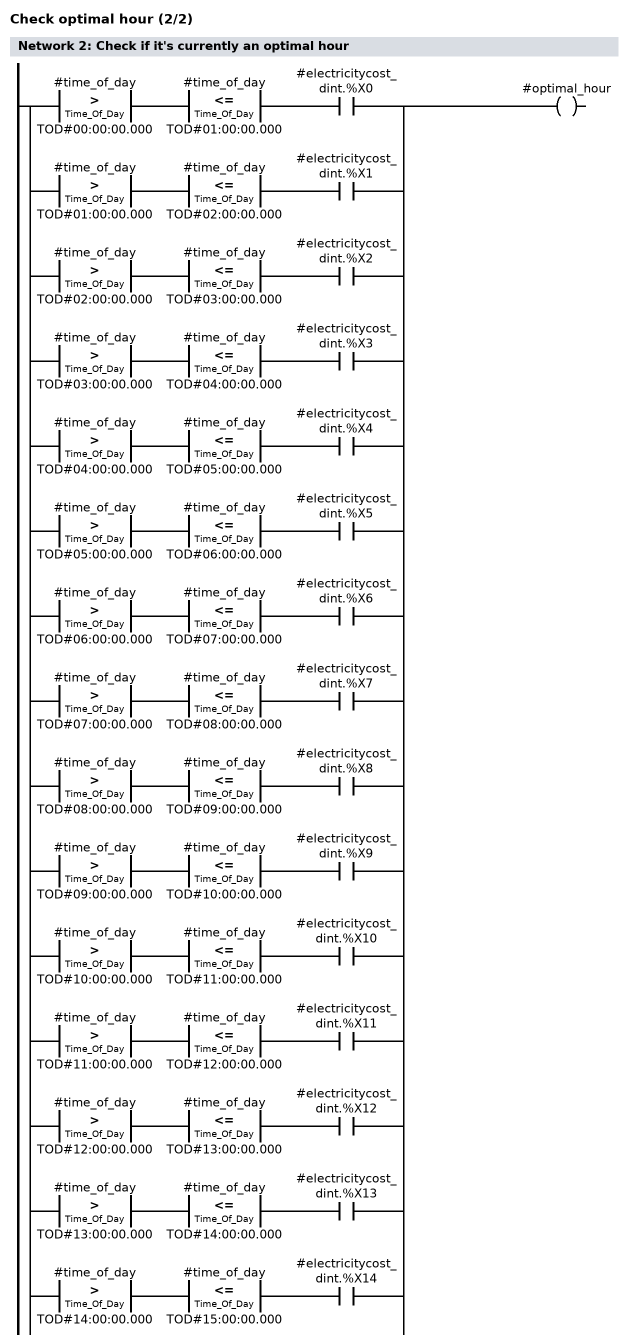
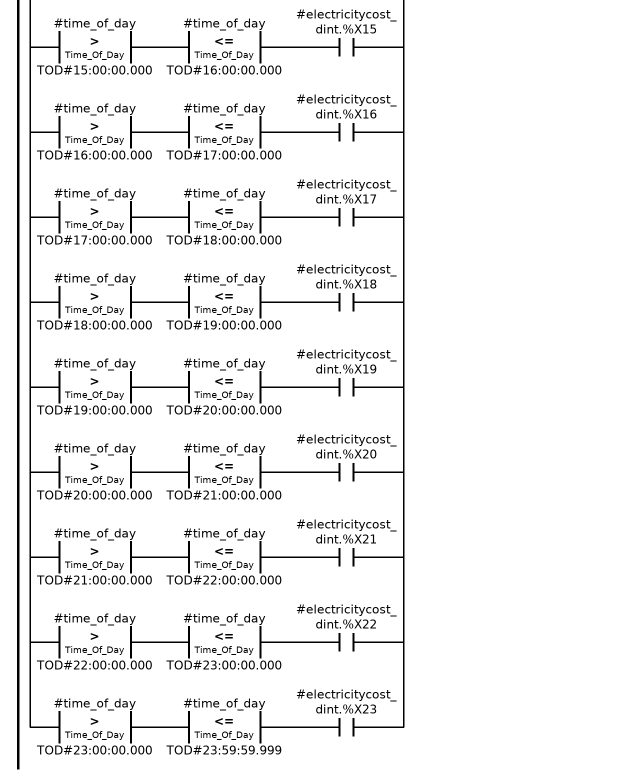
   RUNG wire#powerrail
      { S7_Templates := "SrcType := Time_Of_Day" } GT_Contact(in1 := #time_of_day, in2 := TOD#00:00:00.000)
      { S7_Templates := "SrcType := Time_Of_Day" } LE_Contact(in1 := #time_of_day, in2 := TOD#01:00:00.000)
      Contact( #electricitycost_dint.%X0 )
      wire#w1
      Coil( #optimal_hour )
   END_RUNG
   RUNG wire#powerrail
      { S7_Templates := "SrcType := Time_Of_Day" } GT_Contact(in1 := #time_of_day, in2 := TOD#01:00:00.000)
      { S7_Templates := "SrcType := Time_Of_Day" } LE_Contact(in1 := #time_of_day, in2 := TOD#02:00:00.000)
      Contact( #electricitycost_dint.%X1 )
   END_RUNG wire#w1
   RUNG wire#powerrail
      { S7_Templates := "SrcType := Time_Of_Day" } GT_Contact(in1 := #time_of_day, in2 := TOD#02:00:00.000)
      { S7_Templates := "SrcType := Time_Of_Day" } LE_Contact(in1 := #time_of_day, in2 := TOD#03:00:00.000)
      Contact( #electricitycost_dint.%X2 )
   END_RUNG wire#w1
   RUNG wire#powerrail
      { S7_Templates := "SrcType := Time_Of_Day" } GT_Contact(in1 := #time_of_day, in2 := TOD#03:00:00.000)
      { S7_Templates := "SrcType := Time_Of_Day" } LE_Contact(in1 := #time_of_day, in2 := TOD#04:00:00.000)
      Contact( #electricitycost_dint.%X3 )
   END_RUNG wire#w1
   RUNG wire#powerrail
      { S7_Templates := "SrcType := Time_Of_Day" } GT_Contact(in1 := #time_of_day, in2 := TOD#04:00:00.000)
      { S7_Templates := "SrcType := Time_Of_Day" } LE_Contact(in1 := #time_of_day, in2 := TOD#05:00:00.000)
      Contact( #electricitycost_dint.%X4 )
   END_RUNG wire#w1
   RUNG wire#powerrail
      { S7_Templates := "SrcType := Time_Of_Day" } GT_Contact(in1 := #time_of_day, in2 := TOD#05:00:00.000)
      { S7_Templates := "SrcType := Time_Of_Day" } LE_Contact(in1 := #time_of_day, in2 := TOD#06:00:00.000)
      Contact( #electricitycost_dint.%X5 )
   END_RUNG wire#w1
   RUNG wire#powerrail
      { S7_Templates := "SrcType := Time_Of_Day" } GT_Contact(in1 := #time_of_day, in2 := TOD#06:00:00.000)
      { S7_Templates := "SrcType := Time_Of_Day" } LE_Contact(in1 := #time_of_day, in2 := TOD#07:00:00.000)
      Contact( #electricitycost_dint.%X6 )
   END_RUNG wire#w1
   RUNG wire#powerrail
      { S7_Templates := "SrcType := Time_Of_Day" } GT_Contact(in1 := #time_of_day, in2 := TOD#07:00:00.000)
      { S7_Templates := "SrcType := Time_Of_Day" } LE_Contact(in1 := #time_of_day, in2 := TOD#08:00:00.000)
      Contact( #electricitycost_dint.%X7 )
   END_RUNG wire#w1
   RUNG wire#powerrail
      { S7_Templates := "SrcType := Time_Of_Day" } GT_Contact(in1 := #time_of_day, in2 := TOD#08:00:00.000)
      { S7_Templates := "SrcType := Time_Of_Day" } LE_Contact(in1 := #time_of_day, in2 := TOD#09:00:00.000)
      Contact( #electricitycost_dint.%X8 )
   END_RUNG wire#w1
   RUNG wire#powerrail
      { S7_Templates := "SrcType := Time_Of_Day" } GT_Contact(in1 := #time_of_day, in2 := TOD#09:00:00.000)
      { S7_Templates := "SrcType := Time_Of_Day" } LE_Contact(in1 := #time_of_day, in2 := TOD#10:00:00.000)
      Contact( #electricitycost_dint.%X9 )
   END_RUNG wire#w1
   RUNG wire#powerrail
      { S7_Templates := "SrcType := Time_Of_Day" } GT_Contact(in1 := #time_of_day, in2 := TOD#10:00:00.000)
      { S7_Templates := "SrcType := Time_Of_Day" } LE_Contact(in1 := #time_of_day, in2 := TOD#11:00:00.000)
      Contact( #electricitycost_dint.%X10 )
   END_RUNG wire#w1
   RUNG wire#powerrail
      { S7_Templates := "SrcType := Time_Of_Day" } GT_Contact(in1 := #time_of_day, in2 := TOD#11:00:00.000)
      { S7_Templates := "SrcType := Time_Of_Day" } LE_Contact(in1 := #time_of_day, in2 := TOD#12:00:00.000)
      Contact( #electricitycost_dint.%X11 )
   END_RUNG wire#w1
   RUNG wire#powerrail
      { S7_Templates := "SrcType := Time_Of_Day" } GT_Contact(in1 := #time_of_day, in2 := TOD#12:00:00.000)
      { S7_Templates := "SrcType := Time_Of_Day" } LE_Contact(in1 := #time_of_day, in2 := TOD#13:00:00.000)
      Contact( #electricitycost_dint.%X12 )
   END_RUNG wire#w1
   RUNG wire#powerrail
      { S7_Templates := "SrcType := Time_Of_Day" } GT_Contact(in1 := #time_of_day, in2 := TOD#13:00:00.000)
      { S7_Templates := "SrcType := Time_Of_Day" } LE_Contact(in1 := #time_of_day, in2 := TOD#14:00:00.000)
      Contact( #electricitycost_dint.%X13 )
   END_RUNG wire#w1
   RUNG wire#powerrail
      { S7_Templates := "SrcType := Time_Of_Day" } GT_Contact(in1 := #time_of_day, in2 := TOD#14:00:00.000)
      { S7_Templates := "SrcType := Time_Of_Day" } LE_Contact(in1 := #time_of_day, in2 := TOD#15:00:00.000)
      Contact( #electricitycost_dint.%X14 )
   END_RUNG wire#w1
   RUNG wire#powerrail
      { S7_Templates := "SrcType := Time_Of_Day" } GT_Contact(in1 := #time_of_day, in2 := TOD#15:00:00.000)
      { S7_Templates := "SrcType := Time_Of_Day" } LE_Contact(in1 := #time_of_day, in2 := TOD#16:00:00.000)
      Contact( #electricitycost_dint.%X15 )
   END_RUNG wire#w1
   RUNG wire#powerrail
      { S7_Templates := "SrcType := Time_Of_Day" } GT_Contact(in1 := #time_of_day, in2 := TOD#16:00:00.000)
      { S7_Templates := "SrcType := Time_Of_Day" } LE_Contact(in1 := #time_of_day, in2 := TOD#17:00:00.000)
      Contact( #electricitycost_dint.%X16 )
   END_RUNG wire#w1
   RUNG wire#powerrail
      { S7_Templates := "SrcType := Time_Of_Day" } GT_Contact(in1 := #time_of_day, in2 := TOD#17:00:00.000)
      { S7_Templates := "SrcType := Time_Of_Day" } LE_Contact(in1 := #time_of_day, in2 := TOD#18:00:00.000)
      Contact( #electricitycost_dint.%X17 )
   END_RUNG wire#w1
   RUNG wire#powerrail
      { S7_Templates := "SrcType := Time_Of_Day" } GT_Contact(in1 := #time_of_day, in2 := TOD#18:00:00.000)
      { S7_Templates := "SrcType := Time_Of_Day" } LE_Contact(in1 := #time_of_day, in2 := TOD#19:00:00.000)
      Contact( #electricitycost_dint.%X18 )
   END_RUNG wire#w1
   RUNG wire#powerrail
      { S7_Templates := "SrcType := Time_Of_Day" } GT_Contact(in1 := #time_of_day, in2 := TOD#19:00:00.000)
      { S7_Templates := "SrcType := Time_Of_Day" } LE_Contact(in1 := #time_of_day, in2 := TOD#20:00:00.000)
      Contact( #electricitycost_dint.%X19 )
   END_RUNG wire#w1
   RUNG wire#powerrail
      { S7_Templates := "SrcType := Time_Of_Day" } GT_Contact(in1 := #time_of_day, in2 := TOD#20:00:00.000)
      { S7_Templates := "SrcType := Time_Of_Day" } LE_Contact(in1 := #time_of_day, in2 := TOD#21:00:00.000)
      Contact( #electricitycost_dint.%X20 )
   END_RUNG wire#w1
   RUNG wire#powerrail
      { S7_Templates := "SrcType := Time_Of_Day" } GT_Contact(in1 := #time_of_day, in2 := TOD#21:00:00.000)
      { S7_Templates := "SrcType := Time_Of_Day" } LE_Contact(in1 := #time_of_day, in2 := TOD#22:00:00.000)
      Contact( #electricitycost_dint.%X21 )
   END_RUNG wire#w1
   RUNG wire#powerrail
      { S7_Templates := "SrcType := Time_Of_Day" } GT_Contact(in1 := #time_of_day, in2 := TOD#22:00:00.000)
      { S7_Templates := "SrcType := Time_Of_Day" } LE_Contact(in1 := #time_of_day, in2 := TOD#23:00:00.000)
      Contact( #electricitycost_dint.%X22 )
   END_RUNG wire#w1
   RUNG wire#powerrail
      { S7_Templates := "SrcType := Time_Of_Day" } GT_Contact(in1 := #time_of_day, in2 := TOD#23:00:00.000)
      { S7_Templates := "SrcType := Time_Of_Day" } LE_Contact(in1 := #time_of_day, in2 := TOD#23:59:59.999)
      Contact( #electricitycost_dint.%X23 )
   END_RUNG wire#w1
   // the same network as SCL:
   #optimal_hour := ((#time_of_day > TOD#00:00:00.000) AND (#time_of_day <= TOD#01:00:00.000) AND #electricitycost_dint.%X0) OR ((#time_of_day > TOD#01:00:00.000) AND (#time_of_day <= TOD#02:00:00.000) AND #electricitycost_dint.%X1) OR ((#time_of_day > TOD#02:00:00.000) AND (#time_of_day <= TOD#03:00:00.000) AND #electricitycost_dint.%X2) OR ((#time_of_day > TOD#03:00:00.000) AND (#time_of_day <= TOD#04:00:00.000) AND #electricitycost_dint.%X3) OR ((#time_of_day > TOD#04:00:00.000) AND (#time_of_day <= TOD#05:00:00.000) AND #electricitycost_dint.%X4) OR ((#time_of_day > TOD#05:00:00.000) AND (#time_of_day <= TOD#06:00:00.000) AND #electricitycost_dint.%X5) OR ((#time_of_day > TOD#06:00:00.000) AND (#time_of_day <= TOD#07:00:00.000) AND #electricitycost_dint.%X6) OR ((#time_of_day > TOD#07:00:00.000) AND (#time_of_day <= TOD#08:00:00.000) AND #electricitycost_dint.%X7) OR ((#time_of_day > TOD#08:00:00.000) AND (#time_of_day <= TOD#09:00:00.000) AND #electricitycost_dint.%X8) OR ((#time_of_day > TOD#09:00:00.000) AND (#time_of_day <= TOD#10:00:00.000) AND #electricitycost_dint.%X9) OR ((#time_of_day > TOD#10:00:00.000) AND (#time_of_day <= TOD#11:00:00.000) AND #electricitycost_dint.%X10) OR ((#time_of_day > TOD#11:00:00.000) AND (#time_of_day <= TOD#12:00:00.000) AND #electricitycost_dint.%X11) OR ((#time_of_day > TOD#12:00:00.000) AND (#time_of_day <= TOD#13:00:00.000) AND #electricitycost_dint.%X12) OR ((#time_of_day > TOD#13:00:00.000) AND (#time_of_day <= TOD#14:00:00.000) AND #electricitycost_dint.%X13) OR ((#time_of_day > TOD#14:00:00.000) AND (#time_of_day <= TOD#15:00:00.000) AND #electricitycost_dint.%X14) OR ((#time_of_day > TOD#15:00:00.000) AND (#time_of_day <= TOD#16:00:00.000) AND #electricitycost_dint.%X15) OR ((#time_of_day > TOD#16:00:00.000) AND (#time_of_day <= TOD#17:00:00.000) AND #electricitycost_dint.%X16) OR ((#time_of_day > TOD#17:00:00.000) AND (#time_of_day <= TOD#18:00:00.000) AND #electricitycost_dint.%X17) OR ((#time_of_day > TOD#18:00:00.000) AND (#time_of_day <= TOD#19:00:00.000) AND #electricitycost_dint.%X18) OR ((#time_of_day > TOD#19:00:00.000) AND (#time_of_day <= TOD#20:00:00.000) AND #electricitycost_dint.%X19) OR ((#time_of_day > TOD#20:00:00.000) AND (#time_of_day <= TOD#21:00:00.000) AND #electricitycost_dint.%X20) OR ((#time_of_day > TOD#21:00:00.000) AND (#time_of_day <= TOD#22:00:00.000) AND #electricitycost_dint.%X21) OR ((#time_of_day > TOD#22:00:00.000) AND (#time_of_day <= TOD#23:00:00.000) AND #electricitycost_dint.%X22) OR ((#time_of_day > TOD#23:00:00.000) AND (#time_of_day <= TOD#23:59:59.999) AND #electricitycost_dint.%X23);
END_REGION
END_FUNCTION

// ===== library: MasterCopy "LIC01" =====

FUNCTION_BLOCK "LIC01"   // FB7, LAD
{ S7_Optimized_Access := 'FALSE' }
VERSION : 0.1
   VAR_INPUT
      Regulator_Gain_Master : Real := 10.0;
      Regulator_Ti_Master : Real := 603.0;
      Regulator_Td_Master : Real;
      Regulator_Gain_Slave : Real := 10.0;
      Regulator_Ti_Slave : Real := 603.0;
      Regulator_Td_Slave : Real;
      Regulator_Setpoint_High : Real := 80.0;
      Regulator_Setpoint_Low : Real := 20.0;
      Master_Input : Real;
      Slave_Input : Real;
      Regulator_Man : Bool;
      Regulator_Mv : Real;
      Regulator_Max : Real := 100.0;
      Regulator_Min : Real := 0.0;
      Regulator_State : Int;
   END_VAR
   VAR_OUTPUT
      CV : Real;
      Master_State : Int;
      Slave_State : Int;
      Regulator_Status : Int;
   END_VAR
   VAR_TEMP
      compact_temp : Real;
      reset_controller : Bool;
   END_VAR
BEGIN

REGION Network 1: PID Values
   // Sets the PID values for the regulator
